LIN {X 0,Y 467.107,Z 376.18,A -85,B 0,C 180,E1 -7634.539,E2 -7634.539} C_VEL
LIN {X 0,Y 467.124,Z 376.451,A -85,B 0,C 180,E1 -7634.607,E2 -7634.607} C_VEL
LIN {X 0,Y 469.476,Z 389.998,A -85,B 0,C 180,E1 -7635.044,E2 -7635.044} C_VEL
LIN {X 0,Y 470.129,Z 395.713,A -85,B 0,C 180,E1 -7635.278,E2 -7635.278} C_VEL
LIN {X 0,Y 469.712,Z 407.365,A -85,B 0,C 180,E1 -7635.818,E2 -7635.818} C_VEL
LIN {X 0,Y 469.278,Z 418.568,A -85,B 0,C 180,E1 -7636.5,E2 -7636.5} C_VEL
LIN {X 0,Y 468.844,Z 429.048,A -85,B 0,C 180,E1 -7637.305,E2 -7637.305} C_VEL
LIN {X 0,Y 468.368,Z 439.611,A -85,B 0,C 180,E1 -7638.312,E2 -7638.312} C_VEL
LIN {X 0,Y 467.876,Z 448.784,A -85,B 0,C 180,E1 -7639.397,E2 -7639.397} C_VEL
LIN {X 0,Y 467.447,Z 457.686,A -85,B 0,C 180,E1 -7640.699,E2 -7640.699} C_VEL
LIN {X 0,Y 467.093,Z 464.847,A -85,B 0,C 180,E1 -7641.999,E2 -7641.999} C_VEL
LIN {X 0,Y 466.908,Z 471.07,A -85,B 0,C 180,E1 -7643.438,E2 -7643.438} C_VEL
LIN {X 0,Y 466.784,Z 475.676,A -85,B 0,C 180,E1 -7644.817,E2 -7644.817} C_VEL
LIN {X 0,Y 466.663,Z 477.957,A -85,B 0,C 180,E1 -7645.681,E2 -7645.681} C_VEL
LIN {X 0,Y 466.695,Z 479.806,A -85,B 0,C 180,E1 -7646.546,E2 -7646.546} C_VEL
LIN {X 0,Y 466.646,Z 481.192,A -85,B 0,C 180,E1 -7647.41,E2 -7647.41} C_VEL
LIN {X 0,Y 466.589,Z 482.785,A -85,B 0,C 180,E1 -7649.137,E2 -7649.137} C_VEL
LIN {X 0,Y 466.57,Z 483,A -85,B 0,C 180,E1 -7650,E2 -7650} C_VEL
LIN {X 0,Y 466.589,Z 482.786,A -85,B 0,C 180,E1 -7650.863,E2 -7650.863} C_VEL
LIN {X 0,Y 466.646,Z 481.196,A -85,B 0,C 180,E1 -7652.589,E2 -7652.589} C_VEL
LIN {X 0,Y 466.695,Z 479.811,A -85,B 0,C 180,E1 -7653.453,E2 -7653.453} C_VEL
LIN {X 0,Y 466.703,Z 476.896,A -85,B 0,C 180,E1 -7654.75,E2 -7654.75} C_VEL
LIN {X 0,Y 466.84,Z 472.949,A -85,B 0,C 180,E1 -7656.049,E2 -7656.049} C_VEL
LIN {X 0,Y 466.998,Z 466.878,A -85,B 0,C 180,E1 -7657.566,E2 -7657.566} C_VEL
LIN {X 0,Y 467.349,Z 460.238,A -85,B 0,C 180,E1 -7658.866,E2 -7658.866} C_VEL
LIN {X 0,Y 467.738,Z 451.996,A -85,B 0,C 180,E1 -7660.168,E2 -7660.168} C_VEL
LIN {X 0,Y 468.133,Z 443.527,A -85,B 0,C 180,E1 -7661.254,E2 -7661.254} C_VEL
LIN {X 0,Y 468.659,Z 433.246,A -85,B 0,C 180,E1 -7662.319,E2 -7662.319} C_VEL
LIN {X 0,Y 469.104,Z 421.661,A -85,B 0,C 180,E1 -7663.284,E2 -7663.284} C_VEL
LIN {X 0,Y 469.629,Z 409.366,A -85,B 0,C 180,E1 -7664.074,E2 -7664.074} C_VEL
LIN {X 0,Y 470.056,Z 397.023,A -85,B 0,C 180,E1 -7664.669,E2 -7664.669} C_VEL
LIN {X 0,Y 469.836,Z 392.579,A -85,B 0,C 180,E1 -7664.85,E2 -7664.85} C_VEL
LIN {X 0,Y 467.621,Z 379.497,A -85,B 0,C 180,E1 -7665.312,E2 -7665.312} C_VEL
LIN {X 0,Y 467.094,Z 376.299,A -85,B 0,C 180,E1 -7665.407,E2 -7665.407} C_VEL
LIN {X 0,Y 467.229,Z 368.194,A -85,B 0,C 180,E1 -7668.623,E2 -7668.623} C_VEL
LIN {X 0,Y 467.418,Z 360.751,A -85,B 0,C 180,E1 -7671.614,E2 -7671.614} C_VEL
LIN {X 0,Y 467.623,Z 353.969,A -85,B 0,C 180,E1 -7674.412,E2 -7674.412} C_VEL
LIN {X 0,Y 467.938,Z 346.089,A -85,B 0,C 180,E1 -7677.747,E2 -7677.747} C_VEL
LIN {X 0,Y 468.177,Z 339.319,A -85,B 0,C 180,E1 -7680.689,E2 -7680.689} C_VEL
LIN {X 0,Y 468.481,Z 332.557,A -85,B 0,C 180,E1 -7683.714,E2 -7683.714} C_VEL
LIN {X 0,Y 468.553,Z 327.839,A -85,B 0,C 180,E1 -7685.907,E2 -7685.907} C_VEL
LIN {X 0,Y 467.811,Z 322.365,A -85,B 0,C 180,E1 -7688.629,E2 -7688.629} C_VEL
LIN {X 0,Y 467.615,Z 321.24,A -85,B 0,C 180,E1 -7689.279,E2 -7689.279} C_VEL
LIN {X 0,Y 467.614,Z 321.241,A -85,B 0,C 180,E1 -7692.57,E2 -7692.57} C_VEL
LIN {X 0,Y 467.564,Z 321.245,A -85,B 0,C 180,E1 -7695.052,E2 -7695.052} C_VEL
LIN {X 0,Y 467.558,Z 321.246,A -85,B 0,C 180,E1 -7698.724,E2 -7698.724} C_VEL
LIN {X 0,Y 467.558,Z 321.243,A -85,B 0,C 180,E1 -7701.955,E2 -7701.955} C_VEL
LIN {X 0,Y 467.561,Z 321.244,A -85,B 0,C 180,E1 -7705.167,E2 -7705.167} C_VEL
LIN {X 0,Y 467.573,Z 321.242,A -85,B 0,C 180,E1 -7708.259,E2 -7708.259} C_VEL
LIN {X 0,Y 467.536,Z 321.245,A -85,B 0,C 180,E1 -7711.248,E2 -7711.248} C_VEL
LIN {X 0,Y 467.584,Z 321.244,A -85,B 0,C 180,E1 -7714.396,E2 -7714.396} C_VEL
LIN {X 0,Y 467.568,Z 321.242,A -85,B 0,C 180,E1 -7716.995,E2 -7716.995} C_VEL
LIN {X 0,Y 467.614,Z 321.239,A -85,B 0,C 180,E1 -7719.777,E2 -7719.777} C_VEL
LIN {X 0,Y 467.597,Z 321.241,A -85,B 0,C 180,E1 -7722.506,E2 -7722.506} C_VEL
LIN {X 0,Y 467.589,Z 321.239,A -85,B 0,C 180,E1 -7725.196,E2 -7725.196} C_VEL
LIN {X 0,Y 467.645,Z 321.235,A -85,B 0,C 180,E1 -7727.854,E2 -7727.854} C_VEL
LIN {X 0,Y 467.672,Z 321.23,A -85,B 0,C 180,E1 -7731.357,E2 -7731.357} C_VEL
LIN {X 0,Y 467.744,Z 321.221,A -85,B 0,C 180,E1 -7733.963,E2 -7733.963} C_VEL
LIN {X 0,Y 467.849,Z 321.208,A -85,B 0,C 180,E1 -7737.417,E2 -7737.417} C_VEL
LIN {X 0,Y 467.866,Z 321.207,A -85,B 0,C 180,E1 -7740,E2 -7740} C_VEL
LIN {X 0,Y 467.849,Z 321.205,A -85,B 0,C 180,E1 -7742.583,E2 -7742.583} C_VEL
LIN {X 0,Y 467.74,Z 321.221,A -85,B 0,C 180,E1 -7746.037,E2 -7746.037} C_VEL
LIN {X 0,Y 467.672,Z 321.23,A -85,B 0,C 180,E1 -7748.643,E2 -7748.643} C_VEL
LIN {X 0,Y 467.645,Z 321.233,A -85,B 0,C 180,E1 -7752.146,E2 -7752.146} C_VEL
LIN {X 0,Y 467.639,Z 321.232,A -85,B 0,C 180,E1 -7755.885,E2 -7755.885} C_VEL
LIN {X 0,Y 467.615,Z 321.238,A -85,B 0,C 180,E1 -7759.308,E2 -7759.308} C_VEL
LIN {X 0,Y 467.526,Z 321.248,A -85,B 0,C 180,E1 -7762.074,E2 -7762.074} C_VEL
LIN {X 0,Y 467.574,Z 321.242,A -85,B 0,C 180,E1 -7764.889,E2 -7764.889} C_VEL
LIN {X 0,Y 467.552,Z 321.244,A -85,B 0,C 180,E1 -7767.774,E2 -7767.774} C_VEL
LIN {X 0,Y 467.557,Z 321.245,A -85,B 0,C 180,E1 -7771.045,E2 -7771.045} C_VEL
LIN {X 0,Y 467.583,Z 321.242,A -85,B 0,C 180,E1 -7774.243,E2 -7774.243} C_VEL
LIN {X 0,Y 467.543,Z 321.247,A -85,B 0,C 180,E1 -7777.188,E2 -7777.188} C_VEL
LIN {X 0,Y 467.551,Z 321.245,A -85,B 0,C 180,E1 -7780.268,E2 -7780.268} C_VEL
LIN {X 0,Y 467.54,Z 321.244,A -85,B 0,C 180,E1 -7783.747,E2 -7783.747} C_VEL
LIN {X 0,Y 467.549,Z 321.247,A -85,B 0,C 180,E1 -7786.256,E2 -7786.256} C_VEL
LIN {X 0,Y 467.581,Z 321.241,A -85,B 0,C 180,E1 -7788.723,E2 -7788.723} C_VEL
LIN {X 0,Y 467.569,Z 321.243,A -85,B 0,C 180,E1 -7791.408,E2 -7791.408} C_VEL
LIN {X 0,Y 467.462,Z 321.257,A -85,B 0,C 180,E1 -7794.278,E2 -7794.278} C_VEL
LIN {X 0,Y 467.518,Z 322.884,A -85,B 0,C 180,E1 -7795.771,E2 -7795.771} C_VEL
LIN {X 0,Y 467.362,Z 327.675,A -85,B 0,C 180,E1 -7799.252,E2 -7799.252} C_VEL
LIN {X 0,Y 467.182,Z 331.852,A -85,B 0,C 180,E1 -7802.204,E2 -7802.204} C_VEL
LIN {X 0,Y 467.124,Z 335.994,A -85,B 0,C 180,E1 -7805.086,E2 -7805.086} C_VEL
LIN {X 0,Y 466.969,Z 340.133,A -85,B 0,C 180,E1 -7807.899,E2 -7807.899} C_VEL
LIN {X 0,Y 466.889,Z 344.326,A -85,B 0,C 180,E1 -7810.661,E2 -7810.661} C_VEL
LIN {X 0,Y 466.806,Z 349.167,A -85,B 0,C 180,E1 -7813.739,E2 -7813.739} C_VEL
LIN {X 0,Y 466.72,Z 350.349,A -85,B 0,C 180,E1 -7814.072,E2 -7814.072} C_VEL
LIN {X 0,Y 466.388,Z 353.156,A -85,B 0,C 180,E1 -7814.423,E2 -7814.423} C_VEL
LIN {X 0,Y 465.742,Z 357.77,A -85,B 0,C 180,E1 -7814.736,E2 -7814.736} C_VEL
LIN {X 0,Y 464.822,Z 363.833,A -85,B 0,C 180,E1 -7814.982,E2 -7814.982} C_VEL
LIN {X 0,Y 463.865,Z 370.07,A -85,B 0,C 180,E1 -7815.197,E2 -7815.197} C_VEL
LIN {X 0,Y 463.117,Z 377.21,A -85,B 0,C 180,E1 -7815.509,E2 -7815.509} C_VEL
LIN {X 0,Y 462.623,Z 388.395,A -85,B 0,C 180,E1 -7816.158,E2 -7816.158} C_VEL
LIN {X 0,Y 462.173,Z 400.091,A -85,B 0,C 180,E1 -7817.043,E2 -7817.043} C_VEL
LIN {X 0,Y 461.618,Z 410.516,A -85,B 0,C 180,E1 -7818.028,E2 -7818.028} C_VEL
LIN {X 0,Y 461.162,Z 419.064,A -85,B 0,C 180,E1 -7819.019,E2 -7819.019} C_VEL
LIN {X 0,Y 460.753,Z 426.936,A -85,B 0,C 180,E1 -7820.12,E2 -7820.12} C_VEL
LIN {X 0,Y 460.337,Z 434.631,A -85,B 0,C 180,E1 -7821.44,E2 -7821.44} C_VEL
LIN {X 0,Y 459.979,Z 441.691,A -85,B 0,C 180,E1 -7822.98,E2 -7822.98} C_VEL
LIN {X 0,Y 459.877,Z 446.391,A -85,B 0,C 180,E1 -7824.3,E2 -7824.3} C_VEL
LIN {X 0,Y 459.687,Z 449.993,A -85,B 0,C 180,E1 -7825.616,E2 -7825.616} C_VEL
LIN {X 0,Y 459.708,Z 451.852,A -85,B 0,C 180,E1 -7826.495,E2 -7826.495} C_VEL
LIN {X 0,Y 459.608,Z 453.256,A -85,B 0,C 180,E1 -7827.371,E2 -7827.371} C_VEL
LIN {X 0,Y 459.523,Z 454.869,A -85,B 0,C 180,E1 -7829.124,E2 -7829.124} C_VEL
LIN {X 0,Y 459.53,Z 455.103,A -85,B 0,C 180,E1 -7830,E2 -7830} C_VEL
LIN {X 0,Y 459.523,Z 454.917,A -85,B 0,C 180,E1 -7830.877,E2 -7830.877} C_VEL
LIN {X 0,Y 459.608,Z 453.367,A -85,B 0,C 180,E1 -7832.63,E2 -7832.63} C_VEL
LIN {X 0,Y 459.708,Z 452.012,A -85,B 0,C 180,E1 -7833.506,E2 -7833.506} C_VEL
LIN {X 0,Y 459.674,Z 449.153,A -85,B 0,C 180,E1 -7834.824,E2 -7834.824} C_VEL
LIN {X 0,Y 459.939,Z 445.267,A -85,B 0,C 180,E1 -7836.14,E2 -7836.14} C_VEL
LIN {X 0,Y 460.051,Z 440.261,A -85,B 0,C 180,E1 -7837.461,E2 -7837.461} C_VEL
LIN {X 0,Y 460.379,Z 433.956,A -85,B 0,C 180,E1 -7838.781,E2 -7838.781} C_VEL
LIN {X 0,Y 460.768,Z 426.061,A -85,B 0,C 180,E1 -7840.103,E2 -7840.103} C_VEL
LIN {X 0,Y 461.175,Z 418.013,A -85,B 0,C 180,E1 -7841.204,E2 -7841.204} C_VEL
LIN {X 0,Y 461.799,Z 408.186,A -85,B 0,C 180,E1 -7842.302,E2 -7842.302} C_VEL
LIN {X 0,Y 462.179,Z 398.523,A -85,B 0,C 180,E1 -7843.185,E2 -7843.185} C_VEL
LIN {X 0,Y 462.632,Z 388.238,A -85,B 0,C 180,E1 -7843.944,E2 -7843.944} C_VEL
LIN {X 0,Y 463.138,Z 376.598,A -85,B 0,C 180,E1 -7844.613,E2 -7844.613} C_VEL
LIN {X 0,Y 463.284,Z 367.958,A -85,B 0,C 180,E1 -7845.007,E2 -7845.007} C_VEL
LIN {X 0,Y 460.888,Z 355.74,A -85,B 0,C 180,E1 -7845.503,E2 -7845.503} C_VEL
LIN {X 0,Y 459.767,Z 350.859,A -85,B 0,C 180,E1 -7845.672,E2 -7845.672} C_VEL
LIN {X 0,Y 459.831,Z 346.077,A -85,B 0,C 180,E1 -7848.721,E2 -7848.721} C_VEL
LIN {X 0,Y 459.901,Z 341.846,A -85,B 0,C 180,E1 -7851.516,E2 -7851.516} C_VEL
LIN {X 0,Y 460.006,Z 337.676,A -85,B 0,C 180,E1 -7854.362,E2 -7854.362} C_VEL
LIN {X 0,Y 460.132,Z 333.012,A -85,B 0,C 180,E1 -7857.639,E2 -7857.639} C_VEL
LIN {X 0,Y 460.26,Z 329.333,A -85,B 0,C 180,E1 -7860.258,E2 -7860.258} C_VEL
LIN {X 0,Y 460.403,Z 325.125,A -85,B 0,C 180,E1 -7863.335,E2 -7863.335} C_VEL
LIN {X 0,Y 460.415,Z 322.298,A -85,B 0,C 180,E1 -7865.454,E2 -7865.454} C_VEL
LIN {X 0,Y 460.497,Z 322.124,A -85,B 0,C 180,E1 -7867.623,E2 -7867.623} C_VEL
LIN {X 0,Y 460.539,Z 322.119,A -85,B 0,C 180,E1 -7870.269,E2 -7870.269} C_VEL
LIN {X 0,Y 460.498,Z 322.124,A -85,B 0,C 180,E1 -7873.375,E2 -7873.375} C_VEL
LIN {X 0,Y 460.494,Z 322.122,A -85,B 0,C 180,E1 -7876.624,E2 -7876.624} C_VEL
LIN {X 0,Y 460.521,Z 322.121,A -85,B 0,C 180,E1 -7879.733,E2 -7879.733} C_VEL
LIN {X 0,Y 460.498,Z 322.123,A -85,B 0,C 180,E1 -7882.523,E2 -7882.523} C_VEL
LIN {X 0,Y 460.546,Z 322.12,A -85,B 0,C 180,E1 -7885.624,E2 -7885.624} C_VEL
LIN {X 0,Y 460.534,Z 322.118,A -85,B 0,C 180,E1 -7888.744,E2 -7888.744} C_VEL
LIN {X 0,Y 460.527,Z 322.118,A -85,B 0,C 180,E1 -7892.266,E2 -7892.266} C_VEL
LIN {X 0,Y 460.521,Z 322.123,A -85,B 0,C 180,E1 -7894.703,E2 -7894.703} C_VEL
LIN {X 0,Y 460.506,Z 322.123,A -85,B 0,C 180,E1 -7897.571,E2 -7897.571} C_VEL
LIN {X 0,Y 460.566,Z 322.114,A -85,B 0,C 180,E1 -7900.384,E2 -7900.384} C_VEL
LIN {X 0,Y 460.559,Z 322.116,A -85,B 0,C 180,E1 -7903.146,E2 -7903.146} C_VEL
LIN {X 0,Y 460.542,Z 322.116,A -85,B 0,C 180,E1 -7905.867,E2 -7905.867} C_VEL
LIN {X 0,Y 460.606,Z 322.111,A -85,B 0,C 180,E1 -7908.559,E2 -7908.559} C_VEL
LIN {X 0,Y 460.691,Z 322.1,A -85,B 0,C 180,E1 -7912.108,E2 -7912.108} C_VEL
LIN {X 0,Y 460.694,Z 322.102,A -85,B 0,C 180,E1 -7914.748,E2 -7914.748} C_VEL
LIN {X 0,Y 460.795,Z 322.083,A -85,B 0,C 180,E1 -7917.377,E2 -7917.377} C_VEL
LIN {X 0,Y 460.84,Z 322.082,A -85,B 0,C 180,E1 -7920,E2 -7920} C_VEL
LIN {X 0,Y 460.794,Z 322.087,A -85,B 0,C 180,E1 -7922.622,E2 -7922.622} C_VEL
LIN {X 0,Y 460.707,Z 322.098,A -85,B 0,C 180,E1 -7926.13,E2 -7926.13} C_VEL
LIN {X 0,Y 460.625,Z 322.107,A -85,B 0,C 180,E1 -7928.776,E2 -7928.776} C_VEL
LIN {X 0,Y 460.604,Z 322.11,A -85,B 0,C 180,E1 -7932.334,E2 -7932.334} C_VEL
LIN {X 0,Y 460.596,Z 322.112,A -85,B 0,C 180,E1 -7935.998,E2 -7935.998} C_VEL
LIN {X 0,Y 460.567,Z 322.115,A -85,B 0,C 180,E1 -7938.902,E2 -7938.902} C_VEL
LIN {X 0,Y 460.512,Z 322.122,A -85,B 0,C 180,E1 -7941.486,E2 -7941.486} C_VEL
LIN {X 0,Y 460.526,Z 322.119,A -85,B 0,C 180,E1 -7944.333,E2 -7944.333} C_VEL
LIN {X 0,Y 460.51,Z 322.122,A -85,B 0,C 180,E1 -7947.248,E2 -7947.248} C_VEL
LIN {X 0,Y 460.5,Z 322.123,A -85,B 0,C 180,E1 -7950.241,E2 -7950.241} C_VEL
LIN {X 0,Y 460.527,Z 322.12,A -85,B 0,C 180,E1 -7953.325,E2 -7953.325} C_VEL
LIN {X 0,Y 460.476,Z 322.126,A -85,B 0,C 180,E1 -7956.53,E2 -7956.53} C_VEL
LIN {X 0,Y 460.502,Z 322.122,A -85,B 0,C 180,E1 -7958.892,E2 -7958.892} C_VEL
LIN {X 0,Y 460.499,Z 322.123,A -85,B 0,C 180,E1 -7961.599,E2 -7961.599} C_VEL
LIN {X 0,Y 460.509,Z 322.126,A -85,B 0,C 180,E1 -7964.59,E2 -7964.59} C_VEL
LIN {X 0,Y 460.522,Z 322.123,A -85,B 0,C 180,E1 -7967.819,E2 -7967.819} C_VEL
LIN {X 0,Y 460.594,Z 322.299,A -85,B 0,C 180,E1 -7970.65,E2 -7970.65} C_VEL
LIN {X 0,Y 461.487,Z 327.991,A -85,B 0,C 180,E1 -7973.564,E2 -7973.564} C_VEL
LIN {X 0,Y 461.51,Z 332.461,A -85,B 0,C 180,E1 -7975.706,E2 -7975.706} C_VEL
LIN {X 0,Y 461.231,Z 339.206,A -85,B 0,C 180,E1 -7978.797,E2 -7978.797} C_VEL
LIN {X 0,Y 460.924,Z 346.84,A -85,B 0,C 180,E1 -7982.173,E2 -7982.173} C_VEL
LIN {X 0,Y 460.606,Z 353.852,A -85,B 0,C 180,E1 -7985.191,E2 -7985.191} C_VEL
LIN {X 0,Y 460.389,Z 360.659,A -85,B 0,C 180,E1 -7988.037,E2 -7988.037} C_VEL
LIN {X 0,Y 460.175,Z 368.613,A -85,B 0,C 180,E1 -7991.293,E2 -7991.293} C_VEL
LIN {X 0,Y 460.04,Z 376.143,A -85,B 0,C 180,E1 -7994.353,E2 -7994.353} C_VEL
LIN {X 0,Y 462.464,Z 390.155,A -85,B 0,C 180,E1 -7994.826,E2 -7994.826} C_VEL
LIN {X 0,Y 463.206,Z 396.8,A -85,B 0,C 180,E1 -7995.109,E2 -7995.109} C_VEL
LIN {X 0,Y 462.727,Z 409.139,A -85,B 0,C 180,E1 -7995.711,E2 -7995.711} C_VEL
LIN {X 0,Y 462.223,Z 421.008,A -85,B 0,C 180,E1 -7996.481,E2 -7996.481} C_VEL
LIN {X 0,Y 461.719,Z 432.146,A -85,B 0,C 180,E1 -7997.409,E2 -7997.409} C_VEL
LIN {X 0,Y 461.259,Z 441.353,A -85,B 0,C 180,E1 -7998.353,E2 -7998.353} C_VEL
LIN {X 0,Y 460.756,Z 450.206,A -85,B 0,C 180,E1 -7999.453,E2 -7999.453} C_VEL
LIN {X 0,Y 460.346,Z 458.842,A -85,B 0,C 180,E1 -8000.775,E2 -8000.775} C_VEL
LIN {X 0,Y 459.98,Z 465.743,A -85,B 0,C 180,E1 -8002.096,E2 -8002.096} C_VEL
LIN {X 0,Y 459.808,Z 471.46,A -85,B 0,C 180,E1 -8003.467,E2 -8003.467} C_VEL
LIN {X 0,Y 459.701,Z 475.619,A -85,B 0,C 180,E1 -8004.737,E2 -8004.737} C_VEL
LIN {X 0,Y 459.58,Z 477.914,A -85,B 0,C 180,E1 -8005.615,E2 -8005.615} C_VEL
LIN {X 0,Y 459.591,Z 479.778,A -85,B 0,C 180,E1 -8006.493,E2 -8006.493} C_VEL
LIN {X 0,Y 459.57,Z 481.175,A -85,B 0,C 180,E1 -8007.37,E2 -8007.37} C_VEL
LIN {X 0,Y 459.494,Z 482.778,A -85,B 0,C 180,E1 -8009.123,E2 -8009.123} C_VEL
LIN {X 0,Y 459.474,Z 482.994,A -85,B 0,C 180,E1 -8010,E2 -8010} C_VEL
LIN {X 0,Y 459.494,Z 482.779,A -85,B 0,C 180,E1 -8010.876,E2 -8010.876} C_VEL
LIN {X 0,Y 459.57,Z 481.179,A -85,B 0,C 180,E1 -8012.629,E2 -8012.629} C_VEL
LIN {X 0,Y 459.591,Z 479.783,A -85,B 0,C 180,E1 -8013.506,E2 -8013.506} C_VEL
LIN {X 0,Y 459.634,Z 476.847,A -85,B 0,C 180,E1 -8014.824,E2 -8014.824} C_VEL
LIN {X 0,Y 459.757,Z 472.873,A -85,B 0,C 180,E1 -8016.142,E2 -8016.142} C_VEL
LIN {X 0,Y 459.928,Z 466.76,A -85,B 0,C 180,E1 -8017.683,E2 -8017.683} C_VEL
LIN {X 0,Y 460.305,Z 460.085,A -85,B 0,C 180,E1 -8019.003,E2 -8019.003} C_VEL
LIN {X 0,Y 460.7,Z 451.799,A -85,B 0,C 180,E1 -8020.325,E2 -8020.325} C_VEL
LIN {X 0,Y 461.144,Z 443.31,A -85,B 0,C 180,E1 -8021.427,E2 -8021.427} C_VEL
LIN {X 0,Y 461.674,Z 433.197,A -85,B 0,C 180,E1 -8022.492,E2 -8022.492} C_VEL
LIN {X 0,Y 462.119,Z 422.733,A -85,B 0,C 180,E1 -8023.387,E2 -8023.387} C_VEL
LIN {X 0,Y 462.648,Z 411.072,A -85,B 0,C 180,E1 -8024.178,E2 -8024.178} C_VEL
LIN {X 0,Y 463.128,Z 399.413,A -85,B 0,C 180,E1 -8024.781,E2 -8024.781} C_VEL
LIN {X 0,Y 462.969,Z 393.828,A -85,B 0,C 180,E1 -8025.022,E2 -8025.022} C_VEL
LIN {X 0,Y 460.806,Z 380.747,A -85,B 0,C 180,E1 -8025.508,E2 -8025.508} C_VEL
LIN {X 0,Y 460.028,Z 376.103,A -85,B 0,C 180,E1 -8025.666,E2 -8025.666} C_VEL
LIN {X 0,Y 460.197,Z 367.545,A -85,B 0,C 180,E1 -8029.121,E2 -8029.121} C_VEL
LIN {X 0,Y 460.424,Z 359.456,A -85,B 0,C 180,E1 -8032.432,E2 -8032.432} C_VEL
LIN {X 0,Y 460.735,Z 351.428,A -85,B 0,C 180,E1 -8035.844,E2 -8035.844} C_VEL
LIN {X 0,Y 460.981,Z 344.842,A -85,B 0,C 180,E1 -8038.7,E2 -8038.7} C_VEL
LIN {X 0,Y 461.246,Z 338.699,A -85,B 0,C 180,E1 -8041.43,E2 -8041.43} C_VEL
LIN {X 0,Y 461.55,Z 331.611,A -85,B 0,C 180,E1 -8044.689,E2 -8044.689} C_VEL
LIN {X 0,Y 461.49,Z 327.978,A -85,B 0,C 180,E1 -8046.435,E2 -8046.435} C_VEL
LIN {X 0,Y 460.593,Z 322.114,A -85,B 0,C 180,E1 -8049.477,E2 -8049.477} C_VEL
LIN {X 0,Y 460.538,Z 322.122,A -85,B 0,C 180,E1 -8052.903,E2 -8052.903} C_VEL
LIN {X 0,Y 460.5,Z 322.124,A -85,B 0,C 180,E1 -8055.83,E2 -8055.83} C_VEL
LIN {X 0,Y 460.511,Z 322.123,A -85,B 0,C 180,E1 -8058.986,E2 -8058.986} C_VEL
LIN {X 0,Y 460.52,Z 322.124,A -85,B 0,C 180,E1 -8062.519,E2 -8062.519} C_VEL
LIN {X 0,Y 460.541,Z 322.118,A -85,B 0,C 180,E1 -8065.623,E2 -8065.623} C_VEL
LIN {X 0,Y 460.529,Z 322.122,A -85,B 0,C 180,E1 -8068.744,E2 -8068.744} C_VEL
LIN {X 0,Y 460.522,Z 322.121,A -85,B 0,C 180,E1 -8072.265,E2 -8072.265} C_VEL
LIN {X 0,Y 460.53,Z 322.119,A -85,B 0,C 180,E1 -8074.704,E2 -8074.704} C_VEL
LIN {X 0,Y 460.503,Z 322.122,A -85,B 0,C 180,E1 -8077.571,E2 -8077.571} C_VEL
LIN {X 0,Y 460.56,Z 322.116,A -85,B 0,C 180,E1 -8080.384,E2 -8080.384} C_VEL
LIN {X 0,Y 460.554,Z 322.116,A -85,B 0,C 180,E1 -8083.146,E2 -8083.146} C_VEL
LIN {X 0,Y 460.537,Z 322.119,A -85,B 0,C 180,E1 -8085.867,E2 -8085.867} C_VEL
LIN {X 0,Y 460.6,Z 322.109,A -85,B 0,C 180,E1 -8088.559,E2 -8088.559} C_VEL
LIN {X 0,Y 460.685,Z 322.1,A -85,B 0,C 180,E1 -8092.108,E2 -8092.108} C_VEL
LIN {X 0,Y 460.696,Z 322.098,A -85,B 0,C 180,E1 -8094.748,E2 -8094.748} C_VEL
LIN {X 0,Y 460.814,Z 322.084,A -85,B 0,C 180,E1 -8097.378,E2 -8097.378} C_VEL
LIN {X 0,Y 460.836,Z 322.083,A -85,B 0,C 180,E1 -8100,E2 -8100} C_VEL
LIN {X 0,Y 460.79,Z 322.084,A -85,B 0,C 180,E1 -8102.623,E2 -8102.623} C_VEL
LIN {X 0,Y 460.705,Z 322.097,A -85,B 0,C 180,E1 -8106.13,E2 -8106.13} C_VEL
LIN {X 0,Y 460.619,Z 322.109,A -85,B 0,C 180,E1 -8108.776,E2 -8108.776} C_VEL
LIN {X 0,Y 460.598,Z 322.11,A -85,B 0,C 180,E1 -8112.335,E2 -8112.335} C_VEL
LIN {X 0,Y 460.59,Z 322.109,A -85,B 0,C 180,E1 -8115.998,E2 -8115.998} C_VEL
LIN {X 0,Y 460.562,Z 322.118,A -85,B 0,C 180,E1 -8118.902,E2 -8118.902} C_VEL
LIN {X 0,Y 460.507,Z 322.122,A -85,B 0,C 180,E1 -8121.486,E2 -8121.486} C_VEL
LIN {X 0,Y 460.52,Z 322.121,A -85,B 0,C 180,E1 -8124.334,E2 -8124.334} C_VEL
LIN {X 0,Y 460.508,Z 322.125,A -85,B 0,C 180,E1 -8127.248,E2 -8127.248} C_VEL
LIN {X 0,Y 460.495,Z 322.121,A -85,B 0,C 180,E1 -8130.241,E2 -8130.241} C_VEL
LIN {X 0,Y 460.522,Z 322.119,A -85,B 0,C 180,E1 -8133.326,E2 -8133.326} C_VEL
LIN {X 0,Y 460.472,Z 322.128,A -85,B 0,C 180,E1 -8136.53,E2 -8136.53} C_VEL
LIN {X 0,Y 460.507,Z 322.122,A -85,B 0,C 180,E1 -8139.865,E2 -8139.865} C_VEL
LIN {X 0,Y 460.473,Z 322.128,A -85,B 0,C 180,E1 -8142.897,E2 -8142.897} C_VEL
LIN {X 0,Y 460.504,Z 322.121,A -85,B 0,C 180,E1 -8145.832,E2 -8145.832} C_VEL
LIN {X 0,Y 460.535,Z 322.119,A -85,B 0,C 180,E1 -8148.991,E2 -8148.991} C_VEL
LIN {X 0,Y 460.539,Z 322.118,A -85,B 0,C 180,E1 -8151.27,E2 -8151.27} C_VEL
LIN {X 0,Y 460.385,Z 322.175,A -85,B 0,C 180,E1 -8154.545,E2 -8154.545} C_VEL
LIN {X 0,Y 460.398,Z 325.568,A -85,B 0,C 180,E1 -8157.096,E2 -8157.096} C_VEL
LIN {X 0,Y 460.262,Z 329.196,A -85,B 0,C 180,E1 -8159.743,E2 -8159.743} C_VEL
LIN {X 0,Y 460.122,Z 333.372,A -85,B 0,C 180,E1 -8162.728,E2 -8162.728} C_VEL
LIN {X 0,Y 460.047,Z 337.537,A -85,B 0,C 180,E1 -8165.641,E2 -8165.641} C_VEL
LIN {X 0,Y 459.907,Z 342.129,A -85,B 0,C 180,E1 -8168.775,E2 -8168.775} C_VEL
LIN {X 0,Y 459.782,Z 347.341,A -85,B 0,C 180,E1 -8172.2,E2 -8172.2} C_VEL
LIN {X 0,Y 459.814,Z 350.87,A -85,B 0,C 180,E1 -8174.429,E2 -8174.429} C_VEL
LIN {X 0,Y 462.721,Z 364.62,A -85,B 0,C 180,E1 -8174.939,E2 -8174.939} C_VEL
LIN {X 0,Y 463.319,Z 369.874,A -85,B 0,C 180,E1 -8175.169,E2 -8175.169} C_VEL
LIN {X 0,Y 463.117,Z 377.21,A -85,B 0,C 180,E1 -8175.509,E2 -8175.509} C_VEL
LIN {X 0,Y 462.311,Z 382.642,A -85,B 0,C 180,E1 -8175.779,E2 -8175.779} C_VEL
LIN {X 0,Y 459.222,Z 391.298,A -85,B 0,C 180,E1 -8176.239,E2 -8176.239} C_VEL
LIN {X 0,Y 456.032,Z 399.557,A -85,B 0,C 180,E1 -8176.794,E2 -8176.794} C_VEL
LIN {X 0,Y 455.075,Z 404.364,A -85,B 0,C 180,E1 -8177.206,E2 -8177.206} C_VEL
LIN {X 0,Y 454.567,Z 413.753,A -85,B 0,C 180,E1 -8178.18,E2 -8178.18} C_VEL
LIN {X 0,Y 454.044,Z 422.597,A -85,B 0,C 180,E1 -8179.296,E2 -8179.296} C_VEL
LIN {X 0,Y 453.543,Z 431.224,A -85,B 0,C 180,E1 -8180.637,E2 -8180.637} C_VEL
LIN {X 0,Y 453.115,Z 438.1,A -85,B 0,C 180,E1 -8181.976,E2 -8181.976} C_VEL
LIN {X 0,Y 452.879,Z 443.572,A -85,B 0,C 180,E1 -8183.308,E2 -8183.308} C_VEL
LIN {X 0,Y 452.697,Z 447.924,A -85,B 0,C 180,E1 -8184.656,E2 -8184.656} C_VEL
LIN {X 0,Y 452.595,Z 450.21,A -85,B 0,C 180,E1 -8185.547,E2 -8185.547} C_VEL
LIN {X 0,Y 452.624,Z 452.068,A -85,B 0,C 180,E1 -8186.44,E2 -8186.44} C_VEL
LIN {X 0,Y 452.535,Z 453.472,A -85,B 0,C 180,E1 -8187.33,E2 -8187.33} C_VEL
LIN {X 0,Y 452.431,Z 455.084,A -85,B 0,C 180,E1 -8189.11,E2 -8189.11} C_VEL
LIN {X 0,Y 452.435,Z 455.319,A -85,B 0,C 180,E1 -8190,E2 -8190} C_VEL
LIN {X 0,Y 452.431,Z 455.132,A -85,B 0,C 180,E1 -8190.89,E2 -8190.89} C_VEL
LIN {X 0,Y 452.535,Z 453.582,A -85,B 0,C 180,E1 -8192.671,E2 -8192.671} C_VEL
LIN {X 0,Y 452.623,Z 452.226,A -85,B 0,C 180,E1 -8193.561,E2 -8193.561} C_VEL
LIN {X 0,Y 452.605,Z 449.367,A -85,B 0,C 180,E1 -8194.9,E2 -8194.9} C_VEL
LIN {X 0,Y 452.864,Z 445.482,A -85,B 0,C 180,E1 -8196.237,E2 -8196.237} C_VEL
LIN {X 0,Y 452.995,Z 440.475,A -85,B 0,C 180,E1 -8197.578,E2 -8197.578} C_VEL
LIN {X 0,Y 453.369,Z 434.169,A -85,B 0,C 180,E1 -8198.918,E2 -8198.918} C_VEL
LIN {X 0,Y 453.768,Z 426.274,A -85,B 0,C 180,E1 -8200.26,E2 -8200.26} C_VEL
LIN {X 0,Y 454.34,Z 416.45,A -85,B 0,C 180,E1 -8201.601,E2 -8201.601} C_VEL
LIN {X 0,Y 454.998,Z 406.369,A -85,B 0,C 180,E1 -8202.693,E2 -8202.693} C_VEL
LIN {X 0,Y 455.401,Z 395.936,A -85,B 0,C 180,E1 -8203.612,E2 -8203.612} C_VEL
LIN {X 0,Y 455.924,Z 384.756,A -85,B 0,C 180,E1 -8204.393,E2 -8204.393} C_VEL
LIN {X 0,Y 456.448,Z 372.184,A -85,B 0,C 180,E1 -8205.06,E2 -8205.06} C_VEL
LIN {X 0,Y 456.073,Z 366.868,A -85,B 0,C 180,E1 -8205.302,E2 -8205.302} C_VEL
LIN {X 0,Y 453.381,Z 354.212,A -85,B 0,C 180,E1 -8205.81,E2 -8205.81} C_VEL
LIN {X 0,Y 452.661,Z 351.063,A -85,B 0,C 180,E1 -8205.922,E2 -8205.922} C_VEL
LIN {X 0,Y 452.771,Z 346.265,A -85,B 0,C 180,E1 -8209.024,E2 -8209.024} C_VEL
LIN {X 0,Y 452.836,Z 342.018,A -85,B 0,C 180,E1 -8211.869,E2 -8211.869} C_VEL
LIN {X 0,Y 452.963,Z 337.835,A -85,B 0,C 180,E1 -8214.766,E2 -8214.766} C_VEL
LIN {X 0,Y 453.08,Z 333.512,A -85,B 0,C 180,E1 -8217.851,E2 -8217.851} C_VEL
LIN {X 0,Y 453.247,Z 329.46,A -85,B 0,C 180,E1 -8220.777,E2 -8220.777} C_VEL
LIN {X 0,Y 453.394,Z 325.223,A -85,B 0,C 180,E1 -8223.919,E2 -8223.919} C_VEL
LIN {X 0,Y 453.391,Z 323.807,A -85,B 0,C 180,E1 -8224.997,E2 -8224.997} C_VEL
LIN {X 0,Y 453.413,Z 323.009,A -85,B 0,C 180,E1 -8226.292,E2 -8226.292} C_VEL
LIN {X 0,Y 453.467,Z 323,A -85,B 0,C 180,E1 -8229.452,E2 -8229.452} C_VEL
LIN {X 0,Y 453.476,Z 323.001,A -85,B 0,C 180,E1 -8231.934,E2 -8231.934} C_VEL
LIN {X 0,Y 453.48,Z 323,A -85,B 0,C 180,E1 -8235.471,E2 -8235.471} C_VEL
LIN {X 0,Y 453.467,Z 323.001,A -85,B 0,C 180,E1 -8239.388,E2 -8239.388} C_VEL
LIN {X 0,Y 453.451,Z 323.002,A -85,B 0,C 180,E1 -8242.81,E2 -8242.81} C_VEL
LIN {X 0,Y 453.475,Z 322.997,A -85,B 0,C 180,E1 -8246.087,E2 -8246.087} C_VEL
LIN {X 0,Y 453.471,Z 323.002,A -85,B 0,C 180,E1 -8249.24,E2 -8249.24} C_VEL
LIN {X 0,Y 453.485,Z 322.996,A -85,B 0,C 180,E1 -8252.294,E2 -8252.294} C_VEL
LIN {X 0,Y 453.486,Z 322.997,A -85,B 0,C 180,E1 -8255.264,E2 -8255.264} C_VEL
LIN {X 0,Y 453.476,Z 322.999,A -85,B 0,C 180,E1 -8258.415,E2 -8258.415} C_VEL
LIN {X 0,Y 453.518,Z 322.996,A -85,B 0,C 180,E1 -8261.008,E2 -8261.008} C_VEL
LIN {X 0,Y 453.565,Z 322.984,A -85,B 0,C 180,E1 -8263.879,E2 -8263.879} C_VEL
LIN {X 0,Y 453.559,Z 322.987,A -85,B 0,C 180,E1 -8267.471,E2 -8267.471} C_VEL
LIN {X 0,Y 453.587,Z 322.986,A -85,B 0,C 180,E1 -8271.086,E2 -8271.086} C_VEL
LIN {X 0,Y 453.674,Z 322.973,A -85,B 0,C 180,E1 -8273.775,E2 -8273.775} C_VEL
LIN {X 0,Y 453.739,Z 322.962,A -85,B 0,C 180,E1 -8277.337,E2 -8277.337} C_VEL
LIN {X 0,Y 453.809,Z 322.958,A -85,B 0,C 180,E1 -8280,E2 -8280} C_VEL
LIN {X 0,Y 453.738,Z 322.966,A -85,B 0,C 180,E1 -8282.663,E2 -8282.663} C_VEL
LIN {X 0,Y 453.674,Z 322.974,A -85,B 0,C 180,E1 -8286.225,E2 -8286.225} C_VEL
LIN {X 0,Y 453.588,Z 322.983,A -85,B 0,C 180,E1 -8288.913,E2 -8288.913} C_VEL
LIN {X 0,Y 453.559,Z 322.986,A -85,B 0,C 180,E1 -8292.529,E2 -8292.529} C_VEL
LIN {X 0,Y 453.54,Z 322.99,A -85,B 0,C 180,E1 -8296.196,E2 -8296.196} C_VEL
LIN {X 0,Y 453.516,Z 322.993,A -85,B 0,C 180,E1 -8299.041,E2 -8299.041} C_VEL
LIN {X 0,Y 453.473,Z 323,A -85,B 0,C 180,E1 -8301.836,E2 -8301.836} C_VEL
LIN {X 0,Y 453.496,Z 322.993,A -85,B 0,C 180,E1 -8304.736,E2 -8304.736} C_VEL
LIN {X 0,Y 453.471,Z 322.998,A -85,B 0,C 180,E1 -8307.946,E2 -8307.946} C_VEL
LIN {X 0,Y 453.47,Z 322.998,A -85,B 0,C 180,E1 -8310.76,E2 -8310.76} C_VEL
LIN {X 0,Y 453.475,Z 323,A -85,B 0,C 180,E1 -8313.913,E2 -8313.913} C_VEL
LIN {X 0,Y 453.468,Z 323,A -85,B 0,C 180,E1 -8317.188,E2 -8317.188} C_VEL
LIN {X 0,Y 453.467,Z 322.997,A -85,B 0,C 180,E1 -8320.612,E2 -8320.612} C_VEL
LIN {X 0,Y 453.479,Z 323.001,A -85,B 0,C 180,E1 -8324.529,E2 -8324.529} C_VEL
LIN {X 0,Y 453.479,Z 323.001,A -85,B 0,C 180,E1 -8328.21,E2 -8328.21} C_VEL
LIN {X 0,Y 453.556,Z 323.172,A -85,B 0,C 180,E1 -8330.414,E2 -8330.414} C_VEL
LIN {X 0,Y 454.484,Z 329.145,A -85,B 0,C 180,E1 -8333.525,E2 -8333.525} C_VEL
LIN {X 0,Y 454.512,Z 333.483,A -85,B 0,C 180,E1 -8335.64,E2 -8335.64} C_VEL
LIN {X 0,Y 454.223,Z 340.277,A -85,B 0,C 180,E1 -8338.807,E2 -8338.807} C_VEL
LIN {X 0,Y 453.871,Z 348.105,A -85,B 0,C 180,E1 -8342.32,E2 -8342.32} C_VEL
LIN {X 0,Y 453.557,Z 354.863,A -85,B 0,C 180,E1 -8345.268,E2 -8345.268} C_VEL
LIN {X 0,Y 453.289,Z 362.427,A -85,B 0,C 180,E1 -8348.477,E2 -8348.477} C_VEL
LIN {X 0,Y 453.123,Z 368.736,A -85,B 0,C 180,E1 -8351.106,E2 -8351.106} C_VEL
LIN {X 0,Y 452.937,Z 375.949,A -85,B 0,C 180,E1 -8354.105,E2 -8354.105} C_VEL
LIN {X 0,Y 455.387,Z 389.936,A -85,B 0,C 180,E1 -8354.585,E2 -8354.585} C_VEL
LIN {X 0,Y 456.342,Z 396.584,A -85,B 0,C 180,E1 -8354.879,E2 -8354.879} C_VEL
LIN {X 0,Y 455.831,Z 408.923,A -85,B 0,C 180,E1 -8355.49,E2 -8355.49} C_VEL
LIN {X 0,Y 455.307,Z 420.786,A -85,B 0,C 180,E1 -8356.271,E2 -8356.271} C_VEL
LIN {X 0,Y 454.782,Z 431.289,A -85,B 0,C 180,E1 -8357.152,E2 -8357.152} C_VEL
LIN {X 0,Y 454.27,Z 441.136,A -85,B 0,C 180,E1 -8358.171,E2 -8358.171} C_VEL
LIN {X 0,Y 453.736,Z 449.989,A -85,B 0,C 180,E1 -8359.288,E2 -8359.288} C_VEL
LIN {X 0,Y 453.311,Z 458.626,A -85,B 0,C 180,E1 -8360.631,E2 -8360.631} C_VEL
LIN {X 0,Y 452.924,Z 465.527,A -85,B 0,C 180,E1 -8361.972,E2 -8361.972} C_VEL
LIN {X 0,Y 452.731,Z 471.626,A -85,B 0,C 180,E1 -8363.469,E2 -8363.469} C_VEL
LIN {X 0,Y 452.567,Z 476.628,A -85,B 0,C 180,E1 -8365.1,E2 -8365.1} C_VEL
LIN {X 0,Y 452.488,Z 479.562,A -85,B 0,C 180,E1 -8366.438,E2 -8366.438} C_VEL
LIN {X 0,Y 452.496,Z 480.96,A -85,B 0,C 180,E1 -8367.329,E2 -8367.329} C_VEL
LIN {X 0,Y 452.403,Z 482.564,A -85,B 0,C 180,E1 -8369.11,E2 -8369.11} C_VEL
LIN {X 0,Y 452.381,Z 482.78,A -85,B 0,C 180,E1 -8370,E2 -8370} C_VEL
LIN {X 0,Y 452.403,Z 482.565,A -85,B 0,C 180,E1 -8370.89,E2 -8370.89} C_VEL
LIN {X 0,Y 452.496,Z 480.964,A -85,B 0,C 180,E1 -8372.67,E2 -8372.67} C_VEL
LIN {X 0,Y 452.488,Z 479.567,A -85,B 0,C 180,E1 -8373.561,E2 -8373.561} C_VEL
LIN {X 0,Y 452.567,Z 476.631,A -85,B 0,C 180,E1 -8374.899,E2 -8374.899} C_VEL
LIN {X 0,Y 452.687,Z 471.804,A -85,B 0,C 180,E1 -8376.481,E2 -8376.481} C_VEL
LIN {X 0,Y 452.926,Z 465.531,A -85,B 0,C 180,E1 -8378.027,E2 -8378.027} C_VEL
LIN {X 0,Y 453.31,Z 458.63,A -85,B 0,C 180,E1 -8379.368,E2 -8379.368} C_VEL
LIN {X 0,Y 453.736,Z 449.995,A -85,B 0,C 180,E1 -8380.711,E2 -8380.711} C_VEL
LIN {X 0,Y 454.294,Z 441.144,A -85,B 0,C 180,E1 -8381.828,E2 -8381.828} C_VEL
LIN {X 0,Y 454.835,Z 431.31,A -85,B 0,C 180,E1 -8382.844,E2 -8382.844} C_VEL
LIN {X 0,Y 455.293,Z 420.799,A -85,B 0,C 180,E1 -8383.728,E2 -8383.728} C_VEL
LIN {X 0,Y 455.846,Z 408.934,A -85,B 0,C 180,E1 -8384.508,E2 -8384.508} C_VEL
LIN {X 0,Y 456.309,Z 396.591,A -85,B 0,C 180,E1 -8385.121,E2 -8385.121} C_VEL
LIN {X 0,Y 454.37,Z 384.012,A -85,B 0,C 180,E1 -8385.642,E2 -8385.642} C_VEL
LIN {X 0,Y 452.952,Z 375.933,A -85,B 0,C 180,E1 -8385.901,E2 -8385.901} C_VEL
LIN {X 0,Y 453.154,Z 367.28,A -85,B 0,C 180,E1 -8389.477,E2 -8389.477} C_VEL
LIN {X 0,Y 453.407,Z 359.337,A -85,B 0,C 180,E1 -8392.799,E2 -8392.799} C_VEL
LIN {X 0,Y 453.685,Z 351.847,A -85,B 0,C 180,E1 -8396.041,E2 -8396.041} C_VEL
LIN {X 0,Y 453.983,Z 344.718,A -85,B 0,C 180,E1 -8399.185,E2 -8399.185} C_VEL
LIN {X 0,Y 454.277,Z 337.967,A -85,B 0,C 180,E1 -8402.257,E2 -8402.257} C_VEL
LIN {X 0,Y 454.568,Z 332.187,A -85,B 0,C 180,E1 -8404.973,E2 -8404.973} C_VEL
LIN {X 0,Y 454.312,Z 327.888,A -85,B 0,C 180,E1 -8407.106,E2 -8407.106} C_VEL
LIN {X 0,Y 453.533,Z 322.994,A -85,B 0,C 180,E1 -8409.732,E2 -8409.732} C_VEL
LIN {X 0,Y 453.477,Z 323.003,A -85,B 0,C 180,E1 -8413.247,E2 -8413.247} C_VEL
LIN {X 0,Y 453.456,Z 323.002,A -85,B 0,C 180,E1 -8415.778,E2 -8415.778} C_VEL
LIN {X 0,Y 453.464,Z 322.997,A -85,B 0,C 180,E1 -8419.412,E2 -8419.412} C_VEL
LIN {X 0,Y 453.463,Z 323,A -85,B 0,C 180,E1 -8422.811,E2 -8422.811} C_VEL
LIN {X 0,Y 453.47,Z 323,A -85,B 0,C 180,E1 -8426.087,E2 -8426.087} C_VEL
LIN {X 0,Y 453.465,Z 322.999,A -85,B 0,C 180,E1 -8429.24,E2 -8429.24} C_VEL
LIN {X 0,Y 453.48,Z 322.999,A -85,B 0,C 180,E1 -8432.294,E2 -8432.294} C_VEL
LIN {X 0,Y 453.491,Z 322.994,A -85,B 0,C 180,E1 -8435.264,E2 -8435.264} C_VEL
LIN {X 0,Y 453.471,Z 322.999,A -85,B 0,C 180,E1 -8438.414,E2 -8438.414} C_VEL
LIN {X 0,Y 453.512,Z 322.993,A -85,B 0,C 180,E1 -8441.008,E2 -8441.008} C_VEL
LIN {X 0,Y 453.559,Z 322.988,A -85,B 0,C 180,E1 -8443.879,E2 -8443.879} C_VEL
LIN {X 0,Y 453.553,Z 322.987,A -85,B 0,C 180,E1 -8447.471,E2 -8447.471} C_VEL
LIN {X 0,Y 453.582,Z 322.984,A -85,B 0,C 180,E1 -8451.086,E2 -8451.086} C_VEL
LIN {X 0,Y 453.675,Z 322.974,A -85,B 0,C 180,E1 -8453.775,E2 -8453.775} C_VEL
LIN {X 0,Y 453.755,Z 322.964,A -85,B 0,C 180,E1 -8457.337,E2 -8457.337} C_VEL
LIN {X 0,Y 453.805,Z 322.959,A -85,B 0,C 180,E1 -8460,E2 -8460} C_VEL
LIN {X 0,Y 453.734,Z 322.963,A -85,B 0,C 180,E1 -8462.663,E2 -8462.663} C_VEL
LIN {X 0,Y 453.671,Z 322.974,A -85,B 0,C 180,E1 -8466.225,E2 -8466.225} C_VEL
LIN {X 0,Y 453.582,Z 322.986,A -85,B 0,C 180,E1 -8468.914,E2 -8468.914} C_VEL
LIN {X 0,Y 453.553,Z 322.988,A -85,B 0,C 180,E1 -8472.529,E2 -8472.529} C_VEL
LIN {X 0,Y 453.535,Z 322.987,A -85,B 0,C 180,E1 -8476.196,E2 -8476.196} C_VEL
LIN {X 0,Y 453.511,Z 322.997,A -85,B 0,C 180,E1 -8479.041,E2 -8479.041} C_VEL
LIN {X 0,Y 453.467,Z 322.999,A -85,B 0,C 180,E1 -8481.837,E2 -8481.837} C_VEL
LIN {X 0,Y 453.491,Z 322.997,A -85,B 0,C 180,E1 -8484.736,E2 -8484.736} C_VEL
LIN {X 0,Y 453.466,Z 322.998,A -85,B 0,C 180,E1 -8487.947,E2 -8487.947} C_VEL
LIN {X 0,Y 453.465,Z 323.002,A -85,B 0,C 180,E1 -8490.761,E2 -8490.761} C_VEL
LIN {X 0,Y 453.471,Z 322.997,A -85,B 0,C 180,E1 -8493.913,E2 -8493.913} C_VEL
LIN {X 0,Y 453.447,Z 323.003,A -85,B 0,C 180,E1 -8497.19,E2 -8497.19} C_VEL
LIN {X 0,Y 453.463,Z 323.001,A -85,B 0,C 180,E1 -8500.613,E2 -8500.613} C_VEL
LIN {X 0,Y 453.453,Z 323.001,A -85,B 0,C 180,E1 -8504.223,E2 -8504.223} C_VEL
LIN {X 0,Y 453.458,Z 322.999,A -85,B 0,C 180,E1 -8507.006,E2 -8507.006} C_VEL
LIN {X 0,Y 453.527,Z 322.992,A -85,B 0,C 180,E1 -8510.556,E2 -8510.556} C_VEL
LIN {X 0,Y 453.393,Z 323.01,A -85,B 0,C 180,E1 -8513.913,E2 -8513.913} C_VEL
LIN {X 0,Y 453.395,Z 323.999,A -85,B 0,C 180,E1 -8515.24,E2 -8515.24} C_VEL
LIN {X 0,Y 453.272,Z 327.918,A -85,B 0,C 180,E1 -8518.187,E2 -8518.187} C_VEL
LIN {X 0,Y 453.148,Z 332.129,A -85,B 0,C 180,E1 -8521.264,E2 -8521.264} C_VEL
LIN {X 0,Y 453.021,Z 336.303,A -85,B 0,C 180,E1 -8524.255,E2 -8524.255} C_VEL
LIN {X 0,Y 452.876,Z 340.468,A -85,B 0,C 180,E1 -8527.173,E2 -8527.173} C_VEL
LIN {X 0,Y 452.765,Z 344.692,A -85,B 0,C 180,E1 -8530.033,E2 -8530.033} C_VEL
LIN {X 0,Y 452.688,Z 348.988,A -85,B 0,C 180,E1 -8532.845,E2 -8532.845} C_VEL
LIN {X 0,Y 452.734,Z 351.055,A -85,B 0,C 180,E1 -8534.17,E2 -8534.17} C_VEL
LIN {X 0,Y 455.9,Z 365.983,A -85,B 0,C 180,E1 -8534.751,E2 -8534.751} C_VEL
LIN {X 0,Y 456.435,Z 371.398,A -85,B 0,C 180,E1 -8534.998,E2 -8534.998} C_VEL
LIN {X 0,Y 456.014,Z 383.318,A -85,B 0,C 180,E1 -8535.611,E2 -8535.611} C_VEL
LIN {X 0,Y 455.507,Z 393.869,A -85,B 0,C 180,E1 -8536.318,E2 -8536.318} C_VEL
LIN {X 0,Y 455.075,Z 404.364,A -85,B 0,C 180,E1 -8537.206,E2 -8537.206} C_VEL
LIN {X 0,Y 454.11,Z 409.11,A -85,B 0,C 180,E1 -8537.65,E2 -8537.65} C_VEL
LIN {X 0,Y 450.843,Z 416.483,A -85,B 0,C 180,E1 -8538.391,E2 -8538.391} C_VEL
LIN {X 0,Y 447.643,Z 423.264,A -85,B 0,C 180,E1 -8539.207,E2 -8539.207} C_VEL
LIN {X 0,Y 446.776,Z 427.084,A -85,B 0,C 180,E1 -8539.763,E2 -8539.763} C_VEL
LIN {X 0,Y 446.306,Z 435.067,A -85,B 0,C 180,E1 -8541.169,E2 -8541.169} C_VEL
LIN {X 0,Y 445.886,Z 442.125,A -85,B 0,C 180,E1 -8542.757,E2 -8542.757} C_VEL
LIN {X 0,Y 445.776,Z 446.824,A -85,B 0,C 180,E1 -8544.119,E2 -8544.119} C_VEL
LIN {X 0,Y 445.511,Z 450.427,A -85,B 0,C 180,E1 -8545.477,E2 -8545.477} C_VEL
LIN {X 0,Y 445.527,Z 452.285,A -85,B 0,C 180,E1 -8546.383,E2 -8546.383} C_VEL
LIN {X 0,Y 445.464,Z 453.687,A -85,B 0,C 180,E1 -8547.288,E2 -8547.288} C_VEL
LIN {X 0,Y 445.341,Z 455.3,A -85,B 0,C 180,E1 -8549.096,E2 -8549.096} C_VEL
LIN {X 0,Y 445.342,Z 455.534,A -85,B 0,C 180,E1 -8550,E2 -8550} C_VEL
LIN {X 0,Y 445.341,Z 455.347,A -85,B 0,C 180,E1 -8550.905,E2 -8550.905} C_VEL
LIN {X 0,Y 445.464,Z 453.796,A -85,B 0,C 180,E1 -8552.713,E2 -8552.713} C_VEL
LIN {X 0,Y 445.525,Z 452.441,A -85,B 0,C 180,E1 -8553.618,E2 -8553.618} C_VEL
LIN {X 0,Y 445.542,Z 449.581,A -85,B 0,C 180,E1 -8554.977,E2 -8554.977} C_VEL
LIN {X 0,Y 445.795,Z 445.696,A -85,B 0,C 180,E1 -8556.336,E2 -8556.336} C_VEL
LIN {X 0,Y 445.964,Z 440.689,A -85,B 0,C 180,E1 -8557.698,E2 -8557.698} C_VEL
LIN {X 0,Y 446.36,Z 434.381,A -85,B 0,C 180,E1 -8559.059,E2 -8559.059} C_VEL
LIN {X 0,Y 446.789,Z 426.486,A -85,B 0,C 180,E1 -8560.422,E2 -8560.422} C_VEL
LIN {X 0,Y 447.384,Z 416.662,A -85,B 0,C 180,E1 -8561.784,E2 -8561.784} C_VEL
LIN {X 0,Y 448.064,Z 406.745,A -85,B 0,C 180,E1 -8562.877,E2 -8562.877} C_VEL
LIN {X 0,Y 448.531,Z 395.274,A -85,B 0,C 180,E1 -8563.895,E2 -8563.895} C_VEL
LIN {X 0,Y 449.065,Z 384.964,A -85,B 0,C 180,E1 -8564.617,E2 -8564.617} C_VEL
LIN {X 0,Y 449.593,Z 372.389,A -85,B 0,C 180,E1 -8565.295,E2 -8565.295} C_VEL
LIN {X 0,Y 449.233,Z 368.051,A -85,B 0,C 180,E1 -8565.502,E2 -8565.502} C_VEL
LIN {X 0,Y 446.562,Z 355.376,A -85,B 0,C 180,E1 -8566.033,E2 -8566.033} C_VEL
LIN {X 0,Y 445.583,Z 351.263,A -85,B 0,C 180,E1 -8566.184,E2 -8566.184} C_VEL
LIN {X 0,Y 445.687,Z 346.454,A -85,B 0,C 180,E1 -8569.338,E2 -8569.338} C_VEL
LIN {X 0,Y 445.776,Z 342.192,A -85,B 0,C 180,E1 -8572.233,E2 -8572.233} C_VEL
LIN {X 0,Y 445.906,Z 337.995,A -85,B 0,C 180,E1 -8575.186,E2 -8575.186} C_VEL
LIN {X 0,Y 446.04,Z 333.82,A -85,B 0,C 180,E1 -8578.209,E2 -8578.209} C_VEL
LIN {X 0,Y 446.213,Z 329.587,A -85,B 0,C 180,E1 -8581.316,E2 -8581.316} C_VEL
LIN {X 0,Y 446.352,Z 325.338,A -85,B 0,C 180,E1 -8584.53,E2 -8584.53} C_VEL
LIN {X 0,Y 446.325,Z 323.923,A -85,B 0,C 180,E1 -8585.634,E2 -8585.634} C_VEL
LIN {X 0,Y 446.437,Z 323.877,A -85,B 0,C 180,E1 -8589.027,E2 -8589.027} C_VEL
LIN {X 0,Y 446.434,Z 323.875,A -85,B 0,C 180,E1 -8592.277,E2 -8592.277} C_VEL
LIN {X 0,Y 446.449,Z 323.872,A -85,B 0,C 180,E1 -8595.104,E2 -8595.104} C_VEL
LIN {X 0,Y 446.398,Z 323.878,A -85,B 0,C 180,E1 -8598.605,E2 -8598.605} C_VEL
LIN {X 0,Y 446.41,Z 323.879,A -85,B 0,C 180,E1 -8601.921,E2 -8601.921} C_VEL
LIN {X 0,Y 446.428,Z 323.879,A -85,B 0,C 180,E1 -8605.477,E2 -8605.477} C_VEL
LIN {X 0,Y 446.411,Z 323.877,A -85,B 0,C 180,E1 -8608.699,E2 -8608.699} C_VEL
LIN {X 0,Y 446.422,Z 323.876,A -85,B 0,C 180,E1 -8611.835,E2 -8611.835} C_VEL
LIN {X 0,Y 446.428,Z 323.878,A -85,B 0,C 180,E1 -8614.846,E2 -8614.846} C_VEL
LIN {X 0,Y 446.444,Z 323.874,A -85,B 0,C 180,E1 -8618.245,E2 -8618.245} C_VEL
LIN {X 0,Y 446.452,Z 323.871,A -85,B 0,C 180,E1 -8621.649,E2 -8621.649} C_VEL
LIN {X 0,Y 446.501,Z 323.867,A -85,B 0,C 180,E1 -8624.479,E2 -8624.479} C_VEL
LIN {X 0,Y 446.513,Z 323.866,A -85,B 0,C 180,E1 -8628.193,E2 -8628.193} C_VEL
LIN {X 0,Y 446.596,Z 323.855,A -85,B 0,C 180,E1 -8631.858,E2 -8631.858} C_VEL
LIN {X 0,Y 446.643,Z 323.852,A -85,B 0,C 180,E1 -8634.583,E2 -8634.583} C_VEL
LIN {X 0,Y 446.657,Z 323.849,A -85,B 0,C 180,E1 -8638.197,E2 -8638.197} C_VEL
LIN {X 0,Y 446.779,Z 323.833,A -85,B 0,C 180,E1 -8640,E2 -8640} C_VEL
LIN {X 0,Y 446.685,Z 323.844,A -85,B 0,C 180,E1 -8642.705,E2 -8642.705} C_VEL
LIN {X 0,Y 446.643,Z 323.851,A -85,B 0,C 180,E1 -8646.324,E2 -8646.324} C_VEL
LIN {X 0,Y 446.534,Z 323.861,A -85,B 0,C 180,E1 -8649.055,E2 -8649.055} C_VEL
LIN {X 0,Y 446.517,Z 323.863,A -85,B 0,C 180,E1 -8652.73,E2 -8652.73} C_VEL
LIN {X 0,Y 446.485,Z 323.869,A -85,B 0,C 180,E1 -8656.459,E2 -8656.459} C_VEL
LIN {X 0,Y 446.466,Z 323.872,A -85,B 0,C 180,E1 -8659.303,E2 -8659.303} C_VEL
LIN {X 0,Y 446.415,Z 323.879,A -85,B 0,C 180,E1 -8662.2,E2 -8662.2} C_VEL
LIN {X 0,Y 446.437,Z 323.874,A -85,B 0,C 180,E1 -8665.154,E2 -8665.154} C_VEL
LIN {X 0,Y 446.434,Z 323.874,A -85,B 0,C 180,E1 -8668.182,E2 -8668.182} C_VEL
LIN {X 0,Y 446.411,Z 323.88,A -85,B 0,C 180,E1 -8671.301,E2 -8671.301} C_VEL
LIN {X 0,Y 446.428,Z 323.875,A -85,B 0,C 180,E1 -8674.523,E2 -8674.523} C_VEL
LIN {X 0,Y 446.424,Z 323.875,A -85,B 0,C 180,E1 -8678.081,E2 -8678.081} C_VEL
LIN {X 0,Y 446.397,Z 323.881,A -85,B 0,C 180,E1 -8681.395,E2 -8681.395} C_VEL
LIN {X 0,Y 446.449,Z 323.875,A -85,B 0,C 180,E1 -8685.104,E2 -8685.104} C_VEL
LIN {X 0,Y 446.428,Z 323.877,A -85,B 0,C 180,E1 -8688.609,E2 -8688.609} C_VEL
LIN {X 0,Y 446.499,Z 324.055,A -85,B 0,C 180,E1 -8690.172,E2 -8690.172} C_VEL
LIN {X 0,Y 447.419,Z 329.798,A -85,B 0,C 180,E1 -8693.236,E2 -8693.236} C_VEL
LIN {X 0,Y 447.609,Z 332.773,A -85,B 0,C 180,E1 -8694.732,E2 -8694.732} C_VEL
LIN {X 0,Y 447.252,Z 339.713,A -85,B 0,C 180,E1 -8698.054,E2 -8698.054} C_VEL
LIN {X 0,Y 446.968,Z 345.722,A -85,B 0,C 180,E1 -8700.828,E2 -8700.828} C_VEL
LIN {X 0,Y 446.657,Z 352.489,A -85,B 0,C 180,E1 -8703.86,E2 -8703.86} C_VEL
LIN {X 0,Y 446.334,Z 360.383,A -85,B 0,C 180,E1 -8707.308,E2 -8707.308} C_VEL
LIN {X 0,Y 446.083,Z 368.255,A -85,B 0,C 180,E1 -8710.679,E2 -8710.679} C_VEL
LIN {X 0,Y 445.876,Z 375.721,A -85,B 0,C 180,E1 -8713.844,E2 -8713.844} C_VEL
LIN {X 0,Y 448.373,Z 389.912,A -85,B 0,C 180,E1 -8714.345,E2 -8714.345} C_VEL
LIN {X 0,Y 449.418,Z 397.67,A -85,B 0,C 180,E1 -8714.699,E2 -8714.699} C_VEL
LIN {X 0,Y 448.963,Z 408.708,A -85,B 0,C 180,E1 -8715.263,E2 -8715.263} C_VEL
LIN {X 0,Y 448.398,Z 420.57,A -85,B 0,C 180,E1 -8716.055,E2 -8716.055} C_VEL
LIN {X 0,Y 447.81,Z 431.497,A -85,B 0,C 180,E1 -8716.99,E2 -8716.99} C_VEL
LIN {X 0,Y 447.289,Z 440.92,A -85,B 0,C 180,E1 -8717.984,E2 -8717.984} C_VEL
LIN {X 0,Y 446.72,Z 449.772,A -85,B 0,C 180,E1 -8719.118,E2 -8719.118} C_VEL
LIN {X 0,Y 446.282,Z 458.409,A -85,B 0,C 180,E1 -8720.482,E2 -8720.482} C_VEL
LIN {X 0,Y 445.884,Z 465.311,A -85,B 0,C 180,E1 -8721.844,E2 -8721.844} C_VEL
LIN {X 0,Y 445.658,Z 470.847,A -85,B 0,C 180,E1 -8723.208,E2 -8723.208} C_VEL
LIN {X 0,Y 445.541,Z 475.187,A -85,B 0,C 180,E1 -8724.569,E2 -8724.569} C_VEL
LIN {X 0,Y 445.427,Z 477.483,A -85,B 0,C 180,E1 -8725.475,E2 -8725.475} C_VEL
LIN {X 0,Y 445.387,Z 479.346,A -85,B 0,C 180,E1 -8726.381,E2 -8726.381} C_VEL
LIN {X 0,Y 445.422,Z 480.746,A -85,B 0,C 180,E1 -8727.287,E2 -8727.287} C_VEL
LIN {X 0,Y 445.315,Z 482.349,A -85,B 0,C 180,E1 -8729.095,E2 -8729.095} C_VEL
LIN {X 0,Y 445.292,Z 482.565,A -85,B 0,C 180,E1 -8730,E2 -8730} C_VEL
LIN {X 0,Y 445.315,Z 482.35,A -85,B 0,C 180,E1 -8730.904,E2 -8730.904} C_VEL
LIN {X 0,Y 445.422,Z 480.75,A -85,B 0,C 180,E1 -8732.713,E2 -8732.713} C_VEL
LIN {X 0,Y 445.387,Z 479.352,A -85,B 0,C 180,E1 -8733.618,E2 -8733.618} C_VEL
LIN {X 0,Y 445.5,Z 476.416,A -85,B 0,C 180,E1 -8734.977,E2 -8734.977} C_VEL
LIN {X 0,Y 445.584,Z 472.076,A -85,B 0,C 180,E1 -8736.448,E2 -8736.448} C_VEL
LIN {X 0,Y 445.807,Z 466.328,A -85,B 0,C 180,E1 -8737.928,E2 -8737.928} C_VEL
LIN {X 0,Y 446.193,Z 459.651,A -85,B 0,C 180,E1 -8739.29,E2 -8739.29} C_VEL
LIN {X 0,Y 446.643,Z 451.366,A -85,B 0,C 180,E1 -8740.654,E2 -8740.654} C_VEL
LIN {X 0,Y 447.185,Z 442.878,A -85,B 0,C 180,E1 -8741.788,E2 -8741.788} C_VEL
LIN {X 0,Y 447.744,Z 433.141,A -85,B 0,C 180,E1 -8742.851,E2 -8742.851} C_VEL
LIN {X 0,Y 448.284,Z 422.012,A -85,B 0,C 180,E1 -8743.832,E2 -8743.832} C_VEL
LIN {X 0,Y 448.871,Z 410.64,A -85,B 0,C 180,E1 -8744.623,E2 -8744.623} C_VEL
LIN {X 0,Y 449.378,Z 398.981,A -85,B 0,C 180,E1 -8745.244,E2 -8745.244} C_VEL
LIN {X 0,Y 448.366,Z 389.878,A -85,B 0,C 180,E1 -8745.656,E2 -8745.656} C_VEL
LIN {X 0,Y 446.02,Z 376.988,A -85,B 0,C 180,E1 -8746.118,E2 -8746.118} C_VEL
LIN {X 0,Y 445.882,Z 375.714,A -85,B 0,C 180,E1 -8746.158,E2 -8746.158} C_VEL
LIN {X 0,Y 446.12,Z 367.13,A -85,B 0,C 180,E1 -8749.797,E2 -8749.797} C_VEL
LIN {X 0,Y 446.381,Z 359.245,A -85,B 0,C 180,E1 -8753.178,E2 -8753.178} C_VEL
LIN {X 0,Y 446.687,Z 351.34,A -85,B 0,C 180,E1 -8756.648,E2 -8756.648} C_VEL
LIN {X 0,Y 447.02,Z 344.632,A -85,B 0,C 180,E1 -8759.665,E2 -8759.665} C_VEL
LIN {X 0,Y 447.267,Z 338.974,A -85,B 0,C 180,E1 -8762.292,E2 -8762.292} C_VEL
LIN {X 0,Y 447.609,Z 332.754,A -85,B 0,C 180,E1 -8765.268,E2 -8765.268} C_VEL
LIN {X 0,Y 447.418,Z 329.791,A -85,B 0,C 180,E1 -8766.764,E2 -8766.764} C_VEL
LIN {X 0,Y 446.496,Z 323.871,A -85,B 0,C 180,E1 -8769.92,E2 -8769.92} C_VEL
LIN {X 0,Y 446.442,Z 323.881,A -85,B 0,C 180,E1 -8773.602,E2 -8773.602} C_VEL
LIN {X 0,Y 446.387,Z 323.881,A -85,B 0,C 180,E1 -8776.403,E2 -8776.403} C_VEL
LIN {X 0,Y 446.393,Z 323.877,A -85,B 0,C 180,E1 -8779.796,E2 -8779.796} C_VEL
LIN {X 0,Y 446.418,Z 323.877,A -85,B 0,C 180,E1 -8782.122,E2 -8782.122} C_VEL
LIN {X 0,Y 446.423,Z 323.876,A -85,B 0,C 180,E1 -8785.476,E2 -8785.476} C_VEL
LIN {X 0,Y 446.406,Z 323.881,A -85,B 0,C 180,E1 -8788.699,E2 -8788.699} C_VEL
LIN {X 0,Y 446.437,Z 323.873,A -85,B 0,C 180,E1 -8791.83,E2 -8791.83} C_VEL
LIN {X 0,Y 446.433,Z 323.874,A -85,B 0,C 180,E1 -8794.846,E2 -8794.846} C_VEL
LIN {X 0,Y 446.439,Z 323.876,A -85,B 0,C 180,E1 -8798.244,E2 -8798.244} C_VEL
LIN {X 0,Y 446.447,Z 323.875,A -85,B 0,C 180,E1 -8801.649,E2 -8801.649} C_VEL
LIN {X 0,Y 446.495,Z 323.869,A -85,B 0,C 180,E1 -8804.479,E2 -8804.479} C_VEL
LIN {X 0,Y 446.507,Z 323.867,A -85,B 0,C 180,E1 -8808.193,E2 -8808.193} C_VEL
LIN {X 0,Y 446.59,Z 323.858,A -85,B 0,C 180,E1 -8811.858,E2 -8811.858} C_VEL
LIN {X 0,Y 446.643,Z 323.849,A -85,B 0,C 180,E1 -8814.583,E2 -8814.583} C_VEL
LIN {X 0,Y 446.699,Z 323.843,A -85,B 0,C 180,E1 -8817.295,E2 -8817.295} C_VEL
LIN {X 0,Y 446.775,Z 323.834,A -85,B 0,C 180,E1 -8820,E2 -8820} C_VEL
LIN {X 0,Y 446.682,Z 323.841,A -85,B 0,C 180,E1 -8822.706,E2 -8822.706} C_VEL
LIN {X 0,Y 446.64,Z 323.849,A -85,B 0,C 180,E1 -8826.324,E2 -8826.324} C_VEL
LIN {X 0,Y 446.528,Z 323.866,A -85,B 0,C 180,E1 -8829.056,E2 -8829.056} C_VEL
LIN {X 0,Y 446.511,Z 323.866,A -85,B 0,C 180,E1 -8832.73,E2 -8832.73} C_VEL
LIN {X 0,Y 446.48,Z 323.866,A -85,B 0,C 180,E1 -8836.46,E2 -8836.46} C_VEL
LIN {X 0,Y 446.46,Z 323.873,A -85,B 0,C 180,E1 -8839.304,E2 -8839.304} C_VEL
LIN {X 0,Y 446.409,Z 323.878,A -85,B 0,C 180,E1 -8842.2,E2 -8842.2} C_VEL
LIN {X 0,Y 446.433,Z 323.877,A -85,B 0,C 180,E1 -8845.154,E2 -8845.154} C_VEL
LIN {X 0,Y 446.429,Z 323.875,A -85,B 0,C 180,E1 -8848.183,E2 -8848.183} C_VEL
LIN {X 0,Y 446.406,Z 323.878,A -85,B 0,C 180,E1 -8851.301,E2 -8851.301} C_VEL
LIN {X 0,Y 446.424,Z 323.879,A -85,B 0,C 180,E1 -8854.524,E2 -8854.524} C_VEL
LIN {X 0,Y 446.406,Z 323.879,A -85,B 0,C 180,E1 -8858.08,E2 -8858.08} C_VEL
LIN {X 0,Y 446.398,Z 323.878,A -85,B 0,C 180,E1 -8861.395,E2 -8861.395} C_VEL
LIN {X 0,Y 446.445,Z 323.872,A -85,B 0,C 180,E1 -8865.105,E2 -8865.105} C_VEL
LIN {X 0,Y 446.432,Z 323.876,A -85,B 0,C 180,E1 -8868.611,E2 -8868.611} C_VEL
LIN {X 0,Y 446.468,Z 323.871,A -85,B 0,C 180,E1 -8870.977,E2 -8870.977} C_VEL
LIN {X 0,Y 446.311,Z 323.893,A -85,B 0,C 180,E1 -8874.365,E2 -8874.365} C_VEL
LIN {X 0,Y 446.327,Z 326.646,A -85,B 0,C 180,E1 -8876.57,E2 -8876.57} C_VEL
LIN {X 0,Y 446.162,Z 331.275,A -85,B 0,C 180,E1 -8880.04,E2 -8880.04} C_VEL
LIN {X 0,Y 446.003,Z 335.07,A -85,B 0,C 180,E1 -8882.809,E2 -8882.809} C_VEL
LIN {X 0,Y 445.889,Z 339.643,A -85,B 0,C 180,E1 -8886.091,E2 -8886.091} C_VEL
LIN {X 0,Y 445.726,Z 344.875,A -85,B 0,C 180,E1 -8889.704,E2 -8889.704} C_VEL
LIN {X 0,Y 445.638,Z 349.189,A -85,B 0,C 180,E1 -8892.565,E2 -8892.565} C_VEL
LIN {X 0,Y 445.648,Z 351.311,A -85,B 0,C 180,E1 -8893.922,E2 -8893.922} C_VEL
LIN {X 0,Y 448.502,Z 364.257,A -85,B 0,C 180,E1 -8894.417,E2 -8894.417} C_VEL
LIN {X 0,Y 449.603,Z 371.623,A -85,B 0,C 180,E1 -8894.764,E2 -8894.764} C_VEL
LIN {X 0,Y 449.145,Z 383.541,A -85,B 0,C 180,E1 -8895.386,E2 -8895.386} C_VEL
LIN {X 0,Y 448.546,Z 395.302,A -85,B 0,C 180,E1 -8896.2,E2 -8896.2} C_VEL
LIN {X 0,Y 448.026,Z 406.744,A -85,B 0,C 180,E1 -8897.214,E2 -8897.214} C_VEL
LIN {X 0,Y 447.458,Z 415.917,A -85,B 0,C 180,E1 -8898.219,E2 -8898.219} C_VEL
LIN {X 0,Y 446.962,Z 424.415,A -85,B 0,C 180,E1 -8899.354,E2 -8899.354} C_VEL
LIN {X 0,Y 446.776,Z 427.084,A -85,B 0,C 180,E1 -8899.763,E2 -8899.763} C_VEL
LIN {X 0,Y 445.903,Z 430.761,A -85,B 0,C 180,E1 -8900.346,E2 -8900.346} C_VEL
LIN {X 0,Y 442.695,Z 436.289,A -85,B 0,C 180,E1 -8901.325,E2 -8901.325} C_VEL
LIN {X 0,Y 439.543,Z 441.235,A -85,B 0,C 180,E1 -8902.37,E2 -8902.37} C_VEL
LIN {X 0,Y 438.768,Z 443.857,A -85,B 0,C 180,E1 -8903.052,E2 -8903.052} C_VEL
LIN {X 0,Y 438.606,Z 448.356,A -85,B 0,C 180,E1 -8904.484,E2 -8904.484} C_VEL
LIN {X 0,Y 438.433,Z 450.644,A -85,B 0,C 180,E1 -8905.403,E2 -8905.403} C_VEL
LIN {X 0,Y 438.431,Z 452.501,A -85,B 0,C 180,E1 -8906.324,E2 -8906.324} C_VEL
LIN {X 0,Y 438.395,Z 453.902,A -85,B 0,C 180,E1 -8907.244,E2 -8907.244} C_VEL
LIN {X 0,Y 438.255,Z 455.515,A -85,B 0,C 180,E1 -8909.082,E2 -8909.082} C_VEL
LIN {X 0,Y 438.254,Z 455.749,A -85,B 0,C 180,E1 -8910,E2 -8910} C_VEL
LIN {X 0,Y 438.255,Z 455.562,A -85,B 0,C 180,E1 -8910.919,E2 -8910.919} C_VEL
LIN {X 0,Y 438.395,Z 454.01,A -85,B 0,C 180,E1 -8912.757,E2 -8912.757} C_VEL
LIN {X 0,Y 438.429,Z 452.656,A -85,B 0,C 180,E1 -8913.677,E2 -8913.677} C_VEL
LIN {X 0,Y 438.484,Z 449.795,A -85,B 0,C 180,E1 -8915.058,E2 -8915.058} C_VEL
LIN {X 0,Y 438.71,Z 445.911,A -85,B 0,C 180,E1 -8916.439,E2 -8916.439} C_VEL
LIN {X 0,Y 438.912,Z 440.903,A -85,B 0,C 180,E1 -8917.823,E2 -8917.823} C_VEL
LIN {X 0,Y 439.329,Z 434.595,A -85,B 0,C 180,E1 -8919.205,E2 -8919.205} C_VEL
LIN {X 0,Y 439.816,Z 426.698,A -85,B 0,C 180,E1 -8920.589,E2 -8920.589} C_VEL
LIN {X 0,Y 440.437,Z 416.874,A -85,B 0,C 180,E1 -8921.973,E2 -8921.973} C_VEL
LIN {X 0,Y 441.135,Z 407.091,A -85,B 0,C 180,E1 -8923.069,E2 -8923.069} C_VEL
LIN {X 0,Y 441.61,Z 396.35,A -85,B 0,C 180,E1 -8924.046,E2 -8924.046} C_VEL
LIN {X 0,Y 442.219,Z 385.172,A -85,B 0,C 180,E1 -8924.849,E2 -8924.849} C_VEL
LIN {X 0,Y 442.758,Z 372.594,A -85,B 0,C 180,E1 -8925.537,E2 -8925.537} C_VEL
LIN {X 0,Y 441.4,Z 363.966,A -85,B 0,C 180,E1 -8925.954,E2 -8925.954} C_VEL
LIN {X 0,Y 438.513,Z 351.47,A -85,B 0,C 180,E1 -8926.454,E2 -8926.454} C_VEL
LIN {X 0,Y 438.633,Z 346.642,A -85,B 0,C 180,E1 -8929.662,E2 -8929.662} C_VEL
LIN {X 0,Y 438.713,Z 342.367,A -85,B 0,C 180,E1 -8932.611,E2 -8932.611} C_VEL
LIN {X 0,Y 438.861,Z 338.154,A -85,B 0,C 180,E1 -8935.619,E2 -8935.619} C_VEL
LIN {X 0,Y 439.014,Z 333.963,A -85,B 0,C 180,E1 -8938.702,E2 -8938.702} C_VEL
LIN {X 0,Y 439.194,Z 329.715,A -85,B 0,C 180,E1 -8941.875,E2 -8941.875} C_VEL
LIN {X 0,Y 439.28,Z 326.872,A -85,B 0,C 180,E1 -8944.053,E2 -8944.053} C_VEL
LIN {X 0,Y 439.315,Z 325.249,A -85,B 0,C 180,E1 -8945.325,E2 -8945.325} C_VEL
LIN {X 0,Y 439.334,Z 324.765,A -85,B 0,C 180,E1 -8946.884,E2 -8946.884} C_VEL
LIN {X 0,Y 439.402,Z 324.753,A -85,B 0,C 180,E1 -8949.849,E2 -8949.849} C_VEL
LIN {X 0,Y 439.381,Z 324.752,A -85,B 0,C 180,E1 -8952.626,E2 -8952.626} C_VEL
LIN {X 0,Y 439.396,Z 324.752,A -85,B 0,C 180,E1 -8955.27,E2 -8955.27} C_VEL
LIN {X 0,Y 439.351,Z 324.758,A -85,B 0,C 180,E1 -8959.016,E2 -8959.016} C_VEL
LIN {X 0,Y 439.345,Z 324.758,A -85,B 0,C 180,E1 -8962.564,E2 -8962.564} C_VEL
LIN {X 0,Y 439.399,Z 324.752,A -85,B 0,C 180,E1 -8964.844,E2 -8964.844} C_VEL
LIN {X 0,Y 439.369,Z 324.753,A -85,B 0,C 180,E1 -8968.139,E2 -8968.139} C_VEL
LIN {X 0,Y 439.397,Z 324.751,A -85,B 0,C 180,E1 -8971.606,E2 -8971.606} C_VEL
LIN {X 0,Y 439.368,Z 324.755,A -85,B 0,C 180,E1 -8974.413,E2 -8974.413} C_VEL
LIN {X 0,Y 439.359,Z 324.758,A -85,B 0,C 180,E1 -8977.424,E2 -8977.424} C_VEL
LIN {X 0,Y 439.438,Z 324.747,A -85,B 0,C 180,E1 -8980.663,E2 -8980.663} C_VEL
LIN {X 0,Y 439.457,Z 324.742,A -85,B 0,C 180,E1 -8984.224,E2 -8984.224} C_VEL
LIN {X 0,Y 439.479,Z 324.741,A -85,B 0,C 180,E1 -8988.001,E2 -8988.001} C_VEL
LIN {X 0,Y 439.544,Z 324.733,A -85,B 0,C 180,E1 -8991.726,E2 -8991.726} C_VEL
LIN {X 0,Y 439.618,Z 324.726,A -85,B 0,C 180,E1 -8994.496,E2 -8994.496} C_VEL
LIN {X 0,Y 439.628,Z 324.724,A -85,B 0,C 180,E1 -8998.168,E2 -8998.168} C_VEL
LIN {X 0,Y 439.748,Z 324.709,A -85,B 0,C 180,E1 -9000,E2 -9000} C_VEL
LIN {X 0,Y 439.635,Z 324.723,A -85,B 0,C 180,E1 -9002.749,E2 -9002.749} C_VEL
LIN {X 0,Y 439.614,Z 324.727,A -85,B 0,C 180,E1 -9006.425,E2 -9006.425} C_VEL
LIN {X 0,Y 439.496,Z 324.738,A -85,B 0,C 180,E1 -9009.202,E2 -9009.202} C_VEL
LIN {X 0,Y 439.46,Z 324.741,A -85,B 0,C 180,E1 -9012.938,E2 -9012.938} C_VEL
LIN {X 0,Y 439.443,Z 324.746,A -85,B 0,C 180,E1 -9016.349,E2 -9016.349} C_VEL
LIN {X 0,Y 439.399,Z 324.753,A -85,B 0,C 180,E1 -9019.626,E2 -9019.626} C_VEL
LIN {X 0,Y 439.361,Z 324.755,A -85,B 0,C 180,E1 -9022.576,E2 -9022.576} C_VEL
LIN {X 0,Y 439.374,Z 324.757,A -85,B 0,C 180,E1 -9025.587,E2 -9025.587} C_VEL
LIN {X 0,Y 439.386,Z 324.751,A -85,B 0,C 180,E1 -9028.676,E2 -9028.676} C_VEL
LIN {X 0,Y 439.366,Z 324.756,A -85,B 0,C 180,E1 -9032.031,E2 -9032.031} C_VEL
LIN {X 0,Y 439.393,Z 324.753,A -85,B 0,C 180,E1 -9035.341,E2 -9035.341} C_VEL
LIN {X 0,Y 439.365,Z 324.754,A -85,B 0,C 180,E1 -9038.597,E2 -9038.597} C_VEL
LIN {X 0,Y 439.346,Z 324.756,A -85,B 0,C 180,E1 -9042.21,E2 -9042.21} C_VEL
LIN {X 0,Y 439.397,Z 324.753,A -85,B 0,C 180,E1 -9045.271,E2 -9045.271} C_VEL
LIN {X 0,Y 439.388,Z 324.754,A -85,B 0,C 180,E1 -9048.744,E2 -9048.744} C_VEL
LIN {X 0,Y 439.462,Z 324.929,A -85,B 0,C 180,E1 -9049.923,E2 -9049.923} C_VEL
LIN {X 0,Y 440.345,Z 330.473,A -85,B 0,C 180,E1 -9052.941,E2 -9052.941} C_VEL
LIN {X 0,Y 440.573,Z 334.391,A -85,B 0,C 180,E1 -9054.952,E2 -9054.952} C_VEL
LIN {X 0,Y 440.21,Z 341.104,A -85,B 0,C 180,E1 -9058.207,E2 -9058.207} C_VEL
LIN {X 0,Y 439.847,Z 348.15,A -85,B 0,C 180,E1 -9061.499,E2 -9061.499} C_VEL
LIN {X 0,Y 439.532,Z 354.604,A -85,B 0,C 180,E1 -9064.423,E2 -9064.423} C_VEL
LIN {X 0,Y 439.265,Z 361.34,A -85,B 0,C 180,E1 -9067.419,E2 -9067.419} C_VEL
LIN {X 0,Y 439.007,Z 369.135,A -85,B 0,C 180,E1 -9070.826,E2 -9070.826} C_VEL
LIN {X 0,Y 438.804,Z 375.464,A -85,B 0,C 180,E1 -9073.562,E2 -9073.562} C_VEL
LIN {X 0,Y 441.553,Z 391.245,A -85,B 0,C 180,E1 -9074.157,E2 -9074.157} C_VEL
LIN {X 0,Y 442.508,Z 398.757,A -85,B 0,C 180,E1 -9074.513,E2 -9074.513} C_VEL
LIN {X 0,Y 441.971,Z 410.413,A -85,B 0,C 180,E1 -9075.143,E2 -9075.143} C_VEL
LIN {X 0,Y 441.418,Z 421.784,A -85,B 0,C 180,E1 -9075.948,E2 -9075.948} C_VEL
LIN {X 0,Y 440.748,Z 433.07,A -85,B 0,C 180,E1 -9076.956,E2 -9076.956} C_VEL
LIN {X 0,Y 440.192,Z 442.654,A -85,B 0,C 180,E1 -9078.021,E2 -9078.021} C_VEL
LIN {X 0,Y 439.627,Z 451.144,A -85,B 0,C 180,E1 -9079.173,E2 -9079.173} C_VEL
LIN {X 0,Y 439.166,Z 459.43,A -85,B 0,C 180,E1 -9080.559,E2 -9080.559} C_VEL
LIN {X 0,Y 438.753,Z 466.108,A -85,B 0,C 180,E1 -9081.943,E2 -9081.943} C_VEL
LIN {X 0,Y 438.526,Z 472.224,A -85,B 0,C 180,E1 -9083.558,E2 -9083.558} C_VEL
LIN {X 0,Y 438.415,Z 476.197,A -85,B 0,C 180,E1 -9084.941,E2 -9084.941} C_VEL
LIN {X 0,Y 438.289,Z 479.131,A -85,B 0,C 180,E1 -9086.322,E2 -9086.322} C_VEL
LIN {X 0,Y 438.332,Z 480.53,A -85,B 0,C 180,E1 -9087.243,E2 -9087.243} C_VEL
LIN {X 0,Y 438.23,Z 482.134,A -85,B 0,C 180,E1 -9089.081,E2 -9089.081} C_VEL
LIN {X 0,Y 438.205,Z 482.35,A -85,B 0,C 180,E1 -9090,E2 -9090} C_VEL
LIN {X 0,Y 438.23,Z 482.135,A -85,B 0,C 180,E1 -9090.918,E2 -9090.918} C_VEL
LIN {X 0,Y 438.332,Z 480.534,A -85,B 0,C 180,E1 -9092.757,E2 -9092.757} C_VEL
LIN {X 0,Y 438.289,Z 479.136,A -85,B 0,C 180,E1 -9093.677,E2 -9093.677} C_VEL
LIN {X 0,Y 438.414,Z 476.2,A -85,B 0,C 180,E1 -9095.058,E2 -9095.058} C_VEL
LIN {X 0,Y 438.505,Z 472.224,A -85,B 0,C 180,E1 -9096.441,E2 -9096.441} C_VEL
LIN {X 0,Y 438.754,Z 466.111,A -85,B 0,C 180,E1 -9098.056,E2 -9098.056} C_VEL
LIN {X 0,Y 439.165,Z 459.435,A -85,B 0,C 180,E1 -9099.44,E2 -9099.44} C_VEL
LIN {X 0,Y 439.628,Z 451.149,A -85,B 0,C 180,E1 -9100.826,E2 -9100.826} C_VEL
LIN {X 0,Y 440.212,Z 442.662,A -85,B 0,C 180,E1 -9101.978,E2 -9101.978} C_VEL
LIN {X 0,Y 440.781,Z 433.111,A -85,B 0,C 180,E1 -9103.039,E2 -9103.039} C_VEL
LIN {X 0,Y 441.382,Z 421.796,A -85,B 0,C 180,E1 -9104.052,E2 -9104.052} C_VEL
LIN {X 0,Y 441.98,Z 410.424,A -85,B 0,C 180,E1 -9104.856,E2 -9104.856} C_VEL
LIN {X 0,Y 442.539,Z 398.766,A -85,B 0,C 180,E1 -9105.485,E2 -9105.485} C_VEL
LIN {X 0,Y 440.694,Z 386.083,A -85,B 0,C 180,E1 -9106.059,E2 -9106.059} C_VEL
LIN {X 0,Y 438.803,Z 375.47,A -85,B 0,C 180,E1 -9106.435,E2 -9106.435} C_VEL
LIN {X 0,Y 439.024,Z 368.059,A -85,B 0,C 180,E1 -9109.643,E2 -9109.643} C_VEL
LIN {X 0,Y 439.307,Z 360.231,A -85,B 0,C 180,E1 -9113.075,E2 -9113.075} C_VEL
LIN {X 0,Y 439.652,Z 352.345,A -85,B 0,C 180,E1 -9116.588,E2 -9116.588} C_VEL
LIN {X 0,Y 439.997,Z 345.587,A -85,B 0,C 180,E1 -9119.679,E2 -9119.679} C_VEL
LIN {X 0,Y 440.308,Z 338.858,A -85,B 0,C 180,E1 -9122.866,E2 -9122.866} C_VEL
LIN {X 0,Y 440.608,Z 333.35,A -85,B 0,C 180,E1 -9125.562,E2 -9125.562} C_VEL
LIN {X 0,Y 440.1,Z 328.864,A -85,B 0,C 180,E1 -9127.911,E2 -9127.911} C_VEL
LIN {X 0,Y 439.466,Z 324.748,A -85,B 0,C 180,E1 -9130.227,E2 -9130.227} C_VEL
LIN {X 0,Y 439.389,Z 324.76,A -85,B 0,C 180,E1 -9133.453,E2 -9133.453} C_VEL
LIN {X 0,Y 439.337,Z 324.759,A -85,B 0,C 180,E1 -9136.539,E2 -9136.539} C_VEL
LIN {X 0,Y 439.35,Z 324.759,A -85,B 0,C 180,E1 -9139.016,E2 -9139.016} C_VEL
LIN {X 0,Y 439.366,Z 324.754,A -85,B 0,C 180,E1 -9141.607,E2 -9141.607} C_VEL
LIN {X 0,Y 439.394,Z 324.753,A -85,B 0,C 180,E1 -9144.843,E2 -9144.843} C_VEL
LIN {X 0,Y 439.364,Z 324.757,A -85,B 0,C 180,E1 -9148.139,E2 -9148.139} C_VEL
LIN {X 0,Y 439.391,Z 324.751,A -85,B 0,C 180,E1 -9151.605,E2 -9151.605} C_VEL
LIN {X 0,Y 439.37,Z 324.758,A -85,B 0,C 180,E1 -9154.413,E2 -9154.413} C_VEL
LIN {X 0,Y 439.355,Z 324.756,A -85,B 0,C 180,E1 -9157.424,E2 -9157.424} C_VEL
LIN {X 0,Y 439.432,Z 324.749,A -85,B 0,C 180,E1 -9160.662,E2 -9160.662} C_VEL
LIN {X 0,Y 439.451,Z 324.747,A -85,B 0,C 180,E1 -9164.224,E2 -9164.224} C_VEL
LIN {X 0,Y 439.473,Z 324.746,A -85,B 0,C 180,E1 -9168.001,E2 -9168.001} C_VEL
LIN {X 0,Y 439.538,Z 324.737,A -85,B 0,C 180,E1 -9171.726,E2 -9171.726} C_VEL
LIN {X 0,Y 439.618,Z 324.724,A -85,B 0,C 180,E1 -9174.496,E2 -9174.496} C_VEL
LIN {X 0,Y 439.623,Z 324.725,A -85,B 0,C 180,E1 -9178.168,E2 -9178.168} C_VEL
LIN {X 0,Y 439.744,Z 324.71,A -85,B 0,C 180,E1 -9180,E2 -9180} C_VEL
LIN {X 0,Y 439.631,Z 324.72,A -85,B 0,C 180,E1 -9182.749,E2 -9182.749} C_VEL
LIN {X 0,Y 439.611,Z 324.724,A -85,B 0,C 180,E1 -9186.425,E2 -9186.425} C_VEL
LIN {X 0,Y 439.49,Z 324.742,A -85,B 0,C 180,E1 -9189.202,E2 -9189.202} C_VEL
LIN {X 0,Y 439.455,Z 324.745,A -85,B 0,C 180,E1 -9192.938,E2 -9192.938} C_VEL
LIN {X 0,Y 439.438,Z 324.743,A -85,B 0,C 180,E1 -9196.349,E2 -9196.349} C_VEL
LIN {X 0,Y 439.393,Z 324.752,A -85,B 0,C 180,E1 -9199.627,E2 -9199.627} C_VEL
LIN {X 0,Y 439.355,Z 324.758,A -85,B 0,C 180,E1 -9202.576,E2 -9202.576} C_VEL
LIN {X 0,Y 439.37,Z 324.755,A -85,B 0,C 180,E1 -9205.587,E2 -9205.587} C_VEL
LIN {X 0,Y 439.381,Z 324.754,A -85,B 0,C 180,E1 -9208.676,E2 -9208.676} C_VEL
LIN {X 0,Y 439.361,Z 324.754,A -85,B 0,C 180,E1 -9212.031,E2 -9212.031} C_VEL
LIN {X 0,Y 439.389,Z 324.753,A -85,B 0,C 180,E1 -9215.342,E2 -9215.342} C_VEL
LIN {X 0,Y 439.356,Z 324.758,A -85,B 0,C 180,E1 -9218.598,E2 -9218.598} C_VEL
LIN {X 0,Y 439.351,Z 324.757,A -85,B 0,C 180,E1 -9222.21,E2 -9222.21} C_VEL
LIN {X 0,Y 439.394,Z 324.749,A -85,B 0,C 180,E1 -9225.271,E2 -9225.271} C_VEL
LIN {X 0,Y 439.395,Z 324.752,A -85,B 0,C 180,E1 -9228.743,E2 -9228.743} C_VEL
LIN {X 0,Y 439.378,Z 324.754,A -85,B 0,C 180,E1 -9231.608,E2 -9231.608} C_VEL
LIN {X 0,Y 439.303,Z 324.766,A -85,B 0,C 180,E1 -9233.707,E2 -9233.707} C_VEL
LIN {X 0,Y 439.301,Z 325.326,A -85,B 0,C 180,E1 -9234.836,E2 -9234.836} C_VEL
LIN {X 0,Y 439.241,Z 328.163,A -85,B 0,C 180,E1 -9237.044,E2 -9237.044} C_VEL
LIN {X 0,Y 439.088,Z 332.405,A -85,B 0,C 180,E1 -9240.253,E2 -9240.253} C_VEL
LIN {X 0,Y 438.911,Z 337.107,A -85,B 0,C 180,E1 -9243.727,E2 -9243.727} C_VEL
LIN {X 0,Y 438.799,Z 340.808,A -85,B 0,C 180,E1 -9246.397,E2 -9246.397} C_VEL
LIN {X 0,Y 438.658,Z 345.061,A -85,B 0,C 180,E1 -9249.362,E2 -9249.362} C_VEL
LIN {X 0,Y 438.569,Z 349.388,A -85,B 0,C 180,E1 -9252.274,E2 -9252.274} C_VEL
LIN {X 0,Y 438.539,Z 351.483,A -85,B 0,C 180,E1 -9253.65,E2 -9253.65} C_VEL
LIN {X 0,Y 441.481,Z 364.452,A -85,B 0,C 180,E1 -9254.162,E2 -9254.162} C_VEL
LIN {X 0,Y 442.745,Z 371.85,A -85,B 0,C 180,E1 -9254.522,E2 -9254.522} C_VEL
LIN {X 0,Y 442.274,Z 383.764,A -85,B 0,C 180,E1 -9255.154,E2 -9255.154} C_VEL
LIN {X 0,Y 441.675,Z 395.523,A -85,B 0,C 180,E1 -9255.981,E2 -9255.981} C_VEL
LIN {X 0,Y 441.173,Z 406.079,A -85,B 0,C 180,E1 -9256.924,E2 -9256.924} C_VEL
LIN {X 0,Y 440.519,Z 416.137,A -85,B 0,C 180,E1 -9258.031,E2 -9258.031} C_VEL
LIN {X 0,Y 439.987,Z 424.634,A -85,B 0,C 180,E1 -9259.183,E2 -9259.183} C_VEL
LIN {X 0,Y 439.446,Z 432.888,A -85,B 0,C 180,E1 -9260.566,E2 -9260.566} C_VEL
LIN {X 0,Y 438.981,Z 439.537,A -85,B 0,C 180,E1 -9261.948,E2 -9261.948} C_VEL
LIN {X 0,Y 438.768,Z 443.857,A -85,B 0,C 180,E1 -9263.052,E2 -9263.052} C_VEL
LIN {X 0,Y 438.016,Z 446.287,A -85,B 0,C 180,E1 -9263.748,E2 -9263.748} C_VEL
LIN {X 0,Y 434.993,Z 449.693,A -85,B 0,C 180,E1 -9264.904,E2 -9264.904} C_VEL
LIN {X 0,Y 432.473,Z 451.902,A -85,B 0,C 180,E1 -9265.861,E2 -9265.861} C_VEL
LIN {X 0,Y 431.4,Z 453.27,A -85,B 0,C 180,E1 -9266.614,E2 -9266.614} C_VEL
LIN {X 0,Y 431.317,Z 453.628,A -85,B 0,C 180,E1 -9266.871,E2 -9266.871} C_VEL
LIN {X 0,Y 431.225,Z 455.115,A -85,B 0,C 180,E1 -9268.133,E2 -9268.133} C_VEL
LIN {X 0,Y 431.168,Z 455.964,A -85,B 0,C 180,E1 -9270,E2 -9270} C_VEL
LIN {X 0,Y 431.172,Z 455.777,A -85,B 0,C 180,E1 -9270.934,E2 -9270.934} C_VEL
LIN {X 0,Y 431.327,Z 454.224,A -85,B 0,C 180,E1 -9272.802,E2 -9272.802} C_VEL
LIN {X 0,Y 431.334,Z 452.871,A -85,B 0,C 180,E1 -9273.737,E2 -9273.737} C_VEL
LIN {X 0,Y 431.43,Z 450.009,A -85,B 0,C 180,E1 -9275.141,E2 -9275.141} C_VEL
LIN {X 0,Y 431.656,Z 445.649,A -85,B 0,C 180,E1 -9276.698,E2 -9276.698} C_VEL
LIN {X 0,Y 431.885,Z 441.116,A -85,B 0,C 180,E1 -9277.951,E2 -9277.951} C_VEL
LIN {X 0,Y 432.317,Z 434.808,A -85,B 0,C 180,E1 -9279.356,E2 -9279.356} C_VEL
LIN {X 0,Y 432.846,Z 426.911,A -85,B 0,C 180,E1 -9280.762,E2 -9280.762} C_VEL
LIN {X 0,Y 433.502,Z 417.085,A -85,B 0,C 180,E1 -9282.167,E2 -9282.167} C_VEL
LIN {X 0,Y 434.211,Z 407.453,A -85,B 0,C 180,E1 -9283.266,E2 -9283.266} C_VEL
LIN {X 0,Y 434.719,Z 396.56,A -85,B 0,C 180,E1 -9284.273,E2 -9284.273} C_VEL
LIN {X 0,Y 435.379,Z 385.38,A -85,B 0,C 180,E1 -9285.088,E2 -9285.088} C_VEL
LIN {X 0,Y 435.906,Z 372.799,A -85,B 0,C 180,E1 -9285.788,E2 -9285.788} C_VEL
LIN {X 0,Y 433.564,Z 360.522,A -85,B 0,C 180,E1 -9286.381,E2 -9286.381} C_VEL
LIN {X 0,Y 431.454,Z 351.661,A -85,B 0,C 180,E1 -9286.742,E2 -9286.742} C_VEL
LIN {X 0,Y 431.579,Z 346.833,A -85,B 0,C 180,E1 -9289.997,E2 -9289.997} C_VEL
LIN {X 0,Y 431.662,Z 342.543,A -85,B 0,C 180,E1 -9293.001,E2 -9293.001} C_VEL
LIN {X 0,Y 431.83,Z 338.315,A -85,B 0,C 180,E1 -9296.067,E2 -9296.067} C_VEL
LIN {X 0,Y 431.98,Z 334.107,A -85,B 0,C 180,E1 -9299.214,E2 -9299.214} C_VEL
LIN {X 0,Y 432.172,Z 329.845,A -85,B 0,C 180,E1 -9302.455,E2 -9302.455} C_VEL
LIN {X 0,Y 432.258,Z 326.985,A -85,B 0,C 180,E1 -9304.684,E2 -9304.684} C_VEL
LIN {X 0,Y 432.23,Z 325.647,A -85,B 0,C 180,E1 -9305.828,E2 -9305.828} C_VEL
LIN {X 0,Y 432.337,Z 325.635,A -85,B 0,C 180,E1 -9308.713,E2 -9308.713} C_VEL
LIN {X 0,Y 432.334,Z 325.634,A -85,B 0,C 180,E1 -9311.797,E2 -9311.797} C_VEL
LIN {X 0,Y 432.333,Z 325.629,A -85,B 0,C 180,E1 -9314.347,E2 -9314.347} C_VEL
LIN {X 0,Y 432.3,Z 325.635,A -85,B 0,C 180,E1 -9317.018,E2 -9317.018} C_VEL
LIN {X 0,Y 432.287,Z 325.638,A -85,B 0,C 180,E1 -9319.827,E2 -9319.827} C_VEL
LIN {X 0,Y 432.305,Z 325.637,A -85,B 0,C 180,E1 -9323.022,E2 -9323.022} C_VEL
LIN {X 0,Y 432.358,Z 325.627,A -85,B 0,C 180,E1 -9325.996,E2 -9325.996} C_VEL
LIN {X 0,Y 432.343,Z 325.631,A -85,B 0,C 180,E1 -9329.49,E2 -9329.49} C_VEL
LIN {X 0,Y 432.331,Z 325.63,A -85,B 0,C 180,E1 -9331.873,E2 -9331.873} C_VEL
LIN {X 0,Y 432.372,Z 325.627,A -85,B 0,C 180,E1 -9335.539,E2 -9335.539} C_VEL
LIN {X 0,Y 432.347,Z 325.632,A -85,B 0,C 180,E1 -9339.046,E2 -9339.046} C_VEL
LIN {X 0,Y 432.373,Z 325.624,A -85,B 0,C 180,E1 -9342.011,E2 -9342.011} C_VEL
LIN {X 0,Y 432.388,Z 325.626,A -85,B 0,C 180,E1 -9344.926,E2 -9344.926} C_VEL
LIN {X 0,Y 432.455,Z 325.615,A -85,B 0,C 180,E1 -9347.803,E2 -9347.803} C_VEL
LIN {X 0,Y 432.488,Z 325.611,A -85,B 0,C 180,E1 -9351.59,E2 -9351.59} C_VEL
LIN {X 0,Y 432.594,Z 325.6,A -85,B 0,C 180,E1 -9354.406,E2 -9354.406} C_VEL
LIN {X 0,Y 432.598,Z 325.599,A -85,B 0,C 180,E1 -9358.138,E2 -9358.138} C_VEL
LIN {X 0,Y 432.717,Z 325.585,A -85,B 0,C 180,E1 -9360,E2 -9360} C_VEL
LIN {X 0,Y 432.587,Z 325.601,A -85,B 0,C 180,E1 -9362.794,E2 -9362.794} C_VEL
LIN {X 0,Y 432.569,Z 325.604,A -85,B 0,C 180,E1 -9366.53,E2 -9366.53} C_VEL
LIN {X 0,Y 432.439,Z 325.617,A -85,B 0,C 180,E1 -9369.353,E2 -9369.353} C_VEL
LIN {X 0,Y 432.426,Z 325.617,A -85,B 0,C 180,E1 -9372.803,E2 -9372.803} C_VEL
LIN {X 0,Y 432.408,Z 325.622,A -85,B 0,C 180,E1 -9376.479,E2 -9376.479} C_VEL
LIN {X 0,Y 432.335,Z 325.633,A -85,B 0,C 180,E1 -9379.961,E2 -9379.961} C_VEL
LIN {X 0,Y 432.314,Z 325.633,A -85,B 0,C 180,E1 -9382.965,E2 -9382.965} C_VEL
LIN {X 0,Y 432.334,Z 325.63,A -85,B 0,C 180,E1 -9385.002,E2 -9385.002} C_VEL
LIN {X 0,Y 432.335,Z 325.63,A -85,B 0,C 180,E1 -9388.127,E2 -9388.127} C_VEL
LIN {X 0,Y 432.317,Z 325.636,A -85,B 0,C 180,E1 -9391.346,E2 -9391.346} C_VEL
LIN {X 0,Y 432.338,Z 325.63,A -85,B 0,C 180,E1 -9394.677,E2 -9394.677} C_VEL
LIN {X 0,Y 432.336,Z 325.629,A -85,B 0,C 180,E1 -9398.15,E2 -9398.15} C_VEL
LIN {X 0,Y 432.301,Z 325.634,A -85,B 0,C 180,E1 -9401.801,E2 -9401.801} C_VEL
LIN {X 0,Y 432.331,Z 325.633,A -85,B 0,C 180,E1 -9404.348,E2 -9404.348} C_VEL
LIN {X 0,Y 432.319,Z 325.635,A -85,B 0,C 180,E1 -9407.016,E2 -9407.016} C_VEL
LIN {X 0,Y 432.398,Z 325.81,A -85,B 0,C 180,E1 -9409.668,E2 -9409.668} C_VEL
LIN {X 0,Y 433.278,Z 331.138,A -85,B 0,C 180,E1 -9412.637,E2 -9412.637} C_VEL
LIN {X 0,Y 433.567,Z 335.405,A -85,B 0,C 180,E1 -9414.87,E2 -9414.87} C_VEL
LIN {X 0,Y 433.199,Z 342.102,A -85,B 0,C 180,E1 -9418.18,E2 -9418.18} C_VEL
LIN {X 0,Y 432.845,Z 348.572,A -85,B 0,C 180,E1 -9421.257,E2 -9421.257} C_VEL
LIN {X 0,Y 432.491,Z 355.585,A -85,B 0,C 180,E1 -9424.493,E2 -9424.493} C_VEL
LIN {X 0,Y 432.181,Z 362.307,A -85,B 0,C 180,E1 -9427.534,E2 -9427.534} C_VEL
LIN {X 0,Y 431.932,Z 369.367,A -85,B 0,C 180,E1 -9430.687,E2 -9430.687} C_VEL
LIN {X 0,Y 431.744,Z 375.426,A -85,B 0,C 180,E1 -9433.312,E2 -9433.312} C_VEL
LIN {X 0,Y 434.115,Z 388.768,A -85,B 0,C 180,E1 -9433.789,E2 -9433.789} C_VEL
LIN {X 0,Y 435.612,Z 399.75,A -85,B 0,C 180,E1 -9434.321,E2 -9434.321} C_VEL
LIN {X 0,Y 434.999,Z 411.966,A -85,B 0,C 180,E1 -9435.019,E2 -9435.019} C_VEL
LIN {X 0,Y 434.319,Z 424.421,A -85,B 0,C 180,E1 -9435.952,E2 -9435.952} C_VEL
LIN {X 0,Y 433.621,Z 435.334,A -85,B 0,C 180,E1 -9437.004,E2 -9437.004} C_VEL
LIN {X 0,Y 433.08,Z 444.237,A -85,B 0,C 180,E1 -9438.059,E2 -9438.059} C_VEL
LIN {X 0,Y 432.531,Z 452.42,A -85,B 0,C 180,E1 -9439.23,E2 -9439.23} C_VEL
LIN {X 0,Y 432.066,Z 460.451,A -85,B 0,C 180,E1 -9440.638,E2 -9440.638} C_VEL
LIN {X 0,Y 431.636,Z 466.89,A -85,B 0,C 180,E1 -9442.045,E2 -9442.045} C_VEL
LIN {X 0,Y 431.436,Z 472.32,A -85,B 0,C 180,E1 -9443.555,E2 -9443.555} C_VEL
LIN {X 0,Y 431.288,Z 477.053,A -85,B 0,C 180,E1 -9445.326,E2 -9445.326} C_VEL
LIN {X 0,Y 431.196,Z 478.915,A -85,B 0,C 180,E1 -9446.262,E2 -9446.262} C_VEL
LIN {X 0,Y 431.229,Z 480.314,A -85,B 0,C 180,E1 -9447.197,E2 -9447.197} C_VEL
LIN {X 0,Y 431.199,Z 481.311,A -85,B 0,C 180,E1 -9448.132,E2 -9448.132} C_VEL
LIN {X 0,Y 431.148,Z 481.919,A -85,B 0,C 180,E1 -9449.066,E2 -9449.066} C_VEL
LIN {X 0,Y 431.122,Z 482.135,A -85,B 0,C 180,E1 -9450,E2 -9450} C_VEL
LIN {X 0,Y 431.148,Z 481.92,A -85,B 0,C 180,E1 -9450.934,E2 -9450.934} C_VEL
LIN {X 0,Y 431.199,Z 481.314,A -85,B 0,C 180,E1 -9451.868,E2 -9451.868} C_VEL
LIN {X 0,Y 431.228,Z 480.318,A -85,B 0,C 180,E1 -9452.802,E2 -9452.802} C_VEL
LIN {X 0,Y 431.196,Z 478.92,A -85,B 0,C 180,E1 -9453.738,E2 -9453.738} C_VEL
LIN {X 0,Y 431.33,Z 475.985,A -85,B 0,C 180,E1 -9455.141,E2 -9455.141} C_VEL
LIN {X 0,Y 431.441,Z 472.008,A -85,B 0,C 180,E1 -9456.547,E2 -9456.547} C_VEL
LIN {X 0,Y 431.716,Z 465.896,A -85,B 0,C 180,E1 -9458.189,E2 -9458.189} C_VEL
LIN {X 0,Y 432.137,Z 459.218,A -85,B 0,C 180,E1 -9459.595,E2 -9459.595} C_VEL
LIN {X 0,Y 432.621,Z 450.932,A -85,B 0,C 180,E1 -9461.004,E2 -9461.004} C_VEL
LIN {X 0,Y 433.25,Z 442.445,A -85,B 0,C 180,E1 -9462.173,E2 -9462.173} C_VEL
LIN {X 0,Y 433.87,Z 432.324,A -85,B 0,C 180,E1 -9463.308,E2 -9463.308} C_VEL
LIN {X 0,Y 434.481,Z 421.58,A -85,B 0,C 180,E1 -9464.28,E2 -9464.28} C_VEL
LIN {X 0,Y 435.112,Z 410.208,A -85,B 0,C 180,E1 -9465.096,E2 -9465.096} C_VEL
LIN {X 0,Y 435.563,Z 398.546,A -85,B 0,C 180,E1 -9465.74,E2 -9465.74} C_VEL
LIN {X 0,Y 433.63,Z 385.575,A -85,B 0,C 180,E1 -9466.337,E2 -9466.337} C_VEL
LIN {X 0,Y 431.736,Z 375.25,A -85,B 0,C 180,E1 -9466.71,E2 -9466.71} C_VEL
LIN {X 0,Y 431.979,Z 367.874,A -85,B 0,C 180,E1 -9469.977,E2 -9469.977} C_VEL
LIN {X 0,Y 432.296,Z 360.082,A -85,B 0,C 180,E1 -9473.471,E2 -9473.471} C_VEL
LIN {X 0,Y 432.618,Z 353.001,A -85,B 0,C 180,E1 -9476.685,E2 -9476.685} C_VEL
LIN {X 0,Y 432.96,Z 346.578,A -85,B 0,C 180,E1 -9479.675,E2 -9479.675} C_VEL
LIN {X 0,Y 433.229,Z 340.738,A -85,B 0,C 180,E1 -9482.481,E2 -9482.481} C_VEL
LIN {X 0,Y 433.567,Z 335.4,A -85,B 0,C 180,E1 -9485.13,E2 -9485.13} C_VEL
LIN {X 0,Y 433.276,Z 331.126,A -85,B 0,C 180,E1 -9487.363,E2 -9487.363} C_VEL
LIN {X 0,Y 432.42,Z 325.626,A -85,B 0,C 180,E1 -9490.441,E2 -9490.441} C_VEL
LIN {X 0,Y 432.373,Z 325.629,A -85,B 0,C 180,E1 -9494.341,E2 -9494.341} C_VEL
LIN {X 0,Y 432.302,Z 325.634,A -85,B 0,C 180,E1 -9498.199,E2 -9498.199} C_VEL
LIN {X 0,Y 432.323,Z 325.632,A -85,B 0,C 180,E1 -9501.286,E2 -9501.286} C_VEL
LIN {X 0,Y 432.338,Z 325.634,A -85,B 0,C 180,E1 -9504.367,E2 -9504.367} C_VEL
LIN {X 0,Y 432.315,Z 325.633,A -85,B 0,C 180,E1 -9507.556,E2 -9507.556} C_VEL
LIN {X 0,Y 432.318,Z 325.635,A -85,B 0,C 180,E1 -9510.811,E2 -9510.811} C_VEL
LIN {X 0,Y 432.316,Z 325.633,A -85,B 0,C 180,E1 -9513.964,E2 -9513.964} C_VEL
LIN {X 0,Y 432.358,Z 325.63,A -85,B 0,C 180,E1 -9516.023,E2 -9516.023} C_VEL
LIN {X 0,Y 432.341,Z 325.63,A -85,B 0,C 180,E1 -9519.046,E2 -9519.046} C_VEL
LIN {X 0,Y 432.368,Z 325.629,A -85,B 0,C 180,E1 -9522.011,E2 -9522.011} C_VEL
LIN {X 0,Y 432.382,Z 325.624,A -85,B 0,C 180,E1 -9524.926,E2 -9524.926} C_VEL
LIN {X 0,Y 432.449,Z 325.618,A -85,B 0,C 180,E1 -9527.803,E2 -9527.803} C_VEL
LIN {X 0,Y 432.482,Z 325.615,A -85,B 0,C 180,E1 -9531.59,E2 -9531.59} C_VEL
LIN {X 0,Y 432.594,Z 325.6,A -85,B 0,C 180,E1 -9534.406,E2 -9534.406} C_VEL
LIN {X 0,Y 432.594,Z 325.6,A -85,B 0,C 180,E1 -9538.138,E2 -9538.138} C_VEL
LIN {X 0,Y 432.714,Z 325.585,A -85,B 0,C 180,E1 -9540,E2 -9540} C_VEL
LIN {X 0,Y 432.583,Z 325.598,A -85,B 0,C 180,E1 -9542.794,E2 -9542.794} C_VEL
LIN {X 0,Y 432.565,Z 325.601,A -85,B 0,C 180,E1 -9546.531,E2 -9546.531} C_VEL
LIN {X 0,Y 432.433,Z 325.621,A -85,B 0,C 180,E1 -9549.353,E2 -9549.353} C_VEL
LIN {X 0,Y 432.42,Z 325.621,A -85,B 0,C 180,E1 -9552.804,E2 -9552.804} C_VEL
LIN {X 0,Y 432.403,Z 325.62,A -85,B 0,C 180,E1 -9556.479,E2 -9556.479} C_VEL
LIN {X 0,Y 432.33,Z 325.631,A -85,B 0,C 180,E1 -9559.961,E2 -9559.961} C_VEL
LIN {X 0,Y 432.308,Z 325.636,A -85,B 0,C 180,E1 -9562.965,E2 -9562.965} C_VEL
LIN {X 0,Y 432.33,Z 325.633,A -85,B 0,C 180,E1 -9565.003,E2 -9565.003} C_VEL
LIN {X 0,Y 432.33,Z 325.63,A -85,B 0,C 180,E1 -9568.127,E2 -9568.127} C_VEL
LIN {X 0,Y 432.312,Z 325.633,A -85,B 0,C 180,E1 -9571.347,E2 -9571.347} C_VEL
LIN {X 0,Y 432.334,Z 325.634,A -85,B 0,C 180,E1 -9574.678,E2 -9574.678} C_VEL
LIN {X 0,Y 432.324,Z 325.633,A -85,B 0,C 180,E1 -9578.152,E2 -9578.152} C_VEL
LIN {X 0,Y 432.302,Z 325.634,A -85,B 0,C 180,E1 -9581.801,E2 -9581.801} C_VEL
LIN {X 0,Y 432.328,Z 325.634,A -85,B 0,C 180,E1 -9584.348,E2 -9584.348} C_VEL
LIN {X 0,Y 432.316,Z 325.633,A -85,B 0,C 180,E1 -9587.017,E2 -9587.017} C_VEL
LIN {X 0,Y 432.352,Z 325.629,A -85,B 0,C 180,E1 -9589.818,E2 -9589.818} C_VEL
LIN {X 0,Y 432.29,Z 325.641,A -85,B 0,C 180,E1 -9593.022,E2 -9593.022} C_VEL
LIN {X 0,Y 432.209,Z 325.723,A -85,B 0,C 180,E1 -9594.394,E2 -9594.394} C_VEL
LIN {X 0,Y 432.228,Z 328.287,A -85,B 0,C 180,E1 -9596.439,E2 -9596.439} C_VEL
LIN {X 0,Y 432.082,Z 332.542,A -85,B 0,C 180,E1 -9599.721,E2 -9599.721} C_VEL
LIN {X 0,Y 431.855,Z 336.768,A -85,B 0,C 180,E1 -9602.893,E2 -9602.893} C_VEL
LIN {X 0,Y 431.785,Z 340.979,A -85,B 0,C 180,E1 -9605.99,E2 -9605.99} C_VEL
LIN {X 0,Y 431.592,Z 345.248,A -85,B 0,C 180,E1 -9609.008,E2 -9609.008} C_VEL
LIN {X 0,Y 431.503,Z 349.588,A -85,B 0,C 180,E1 -9611.974,E2 -9611.974} C_VEL
LIN {X 0,Y 431.499,Z 351.814,A -85,B 0,C 180,E1 -9613.38,E2 -9613.38} C_VEL
LIN {X 0,Y 434.501,Z 365.025,A -85,B 0,C 180,E1 -9613.914,E2 -9613.914} C_VEL
LIN {X 0,Y 435.892,Z 373.369,A -85,B 0,C 180,E1 -9614.333,E2 -9614.333} C_VEL
LIN {X 0,Y 435.344,Z 385.773,A -85,B 0,C 180,E1 -9615.032,E2 -9615.032} C_VEL
LIN {X 0,Y 434.731,Z 396.878,A -85,B 0,C 180,E1 -9615.847,E2 -9615.847} C_VEL
LIN {X 0,Y 434.142,Z 408.189,A -85,B 0,C 180,E1 -9616.902,E2 -9616.902} C_VEL
LIN {X 0,Y 433.413,Z 418.168,A -85,B 0,C 180,E1 -9618.069,E2 -9618.069} C_VEL
LIN {X 0,Y 432.766,Z 427.811,A -85,B 0,C 180,E1 -9619.474,E2 -9619.474} C_VEL
LIN {X 0,Y 432.26,Z 435.503,A -85,B 0,C 180,E1 -9620.879,E2 -9620.879} C_VEL
LIN {X 0,Y 431.784,Z 442.561,A -85,B 0,C 180,E1 -9622.519,E2 -9622.519} C_VEL
LIN {X 0,Y 431.632,Z 447.258,A -85,B 0,C 180,E1 -9623.925,E2 -9623.925} C_VEL
LIN {X 0,Y 431.36,Z 450.86,A -85,B 0,C 180,E1 -9625.328,E2 -9625.328} C_VEL
LIN {X 0,Y 431.317,Z 453.628,A -85,B 0,C 180,E1 -9626.871,E2 -9626.871} C_VEL
LIN {X 0,Y 430.64,Z 454.684,A -85,B 0,C 180,E1 -9627.639,E2 -9627.639} C_VEL
LIN {X 0,Y 427.71,Z 455.898,A -85,B 0,C 180,E1 -9628.894,E2 -9628.894} C_VEL
LIN {X 0,Y 425.234,Z 456.265,A -85,B 0,C 180,E1 -9629.913,E2 -9629.913} C_VEL
LIN {X 0,Y 424.174,Z 456.12,A -85,B 0,C 180,E1 -9630.702,E2 -9630.702} C_VEL
LIN {X 0,Y 424.092,Z 455.98,A -85,B 0,C 180,E1 -9630.969,E2 -9630.969} C_VEL
LIN {X 0,Y 424.241,Z 454.439,A -85,B 0,C 180,E1 -9632.849,E2 -9632.849} C_VEL
LIN {X 0,Y 424.241,Z 453.086,A -85,B 0,C 180,E1 -9633.8,E2 -9633.8} C_VEL
LIN {X 0,Y 424.379,Z 450.223,A -85,B 0,C 180,E1 -9635.226,E2 -9635.226} C_VEL
LIN {X 0,Y 424.584,Z 446.197,A -85,B 0,C 180,E1 -9636.702,E2 -9636.702} C_VEL
LIN {X 0,Y 424.854,Z 441.33,A -85,B 0,C 180,E1 -9638.083,E2 -9638.083} C_VEL
LIN {X 0,Y 425.317,Z 435.021,A -85,B 0,C 180,E1 -9639.511,E2 -9639.511} C_VEL
LIN {X 0,Y 425.877,Z 427.123,A -85,B 0,C 180,E1 -9640.94,E2 -9640.94} C_VEL
LIN {X 0,Y 426.423,Z 419.072,A -85,B 0,C 180,E1 -9642.131,E2 -9642.131} C_VEL
LIN {X 0,Y 427.202,Z 409.24,A -85,B 0,C 180,E1 -9643.316,E2 -9643.316} C_VEL
LIN {X 0,Y 427.699,Z 399.573,A -85,B 0,C 180,E1 -9644.27,E2 -9644.27} C_VEL
LIN {X 0,Y 428.311,Z 389.108,A -85,B 0,C 180,E1 -9645.099,E2 -9645.099} C_VEL
LIN {X 0,Y 428.977,Z 376.5,A -85,B 0,C 180,E1 -9645.866,E2 -9645.866} C_VEL
LIN {X 0,Y 428.771,Z 371.717,A -85,B 0,C 180,E1 -9646.119,E2 -9646.119} C_VEL
LIN {X 0,Y 426.238,Z 359.53,A -85,B 0,C 180,E1 -9646.711,E2 -9646.711} C_VEL
LIN {X 0,Y 424.367,Z 351.877,A -85,B 0,C 180,E1 -9647.024,E2 -9647.024} C_VEL
LIN {X 0,Y 424.505,Z 348.456,A -85,B 0,C 180,E1 -9649.337,E2 -9649.337} C_VEL
LIN {X 0,Y 424.58,Z 344.161,A -85,B 0,C 180,E1 -9652.378,E2 -9652.378} C_VEL
LIN {X 0,Y 424.728,Z 339.887,A -85,B 0,C 180,E1 -9655.482,E2 -9655.482} C_VEL
LIN {X 0,Y 424.903,Z 335.534,A -85,B 0,C 180,E1 -9658.761,E2 -9658.761} C_VEL
LIN {X 0,Y 425.091,Z 331.407,A -85,B 0,C 180,E1 -9661.941,E2 -9661.941} C_VEL
LIN {X 0,Y 425.22,Z 328.444,A -85,B 0,C 180,E1 -9664.269,E2 -9664.269} C_VEL
LIN {X 0,Y 425.185,Z 326.525,A -85,B 0,C 180,E1 -9665.91,E2 -9665.91} C_VEL
LIN {X 0,Y 425.278,Z 326.512,A -85,B 0,C 180,E1 -9669.04,E2 -9669.04} C_VEL
LIN {X 0,Y 425.29,Z 326.511,A -85,B 0,C 180,E1 -9671.958,E2 -9671.958} C_VEL
LIN {X 0,Y 425.283,Z 326.51,A -85,B 0,C 180,E1 -9675.283,E2 -9675.283} C_VEL
LIN {X 0,Y 425.245,Z 326.513,A -85,B 0,C 180,E1 -9678.618,E2 -9678.618} C_VEL
LIN {X 0,Y 425.279,Z 326.512,A -85,B 0,C 180,E1 -9681.099,E2 -9681.099} C_VEL
LIN {X 0,Y 425.298,Z 326.507,A -85,B 0,C 180,E1 -9684.664,E2 -9684.664} C_VEL
LIN {X 0,Y 425.262,Z 326.51,A -85,B 0,C 180,E1 -9688.073,E2 -9688.073} C_VEL
LIN {X 0,Y 425.301,Z 326.508,A -85,B 0,C 180,E1 -9691.366,E2 -9691.366} C_VEL
LIN {X 0,Y 425.263,Z 326.513,A -85,B 0,C 180,E1 -9694.552,E2 -9694.552} C_VEL
LIN {X 0,Y 425.299,Z 326.51,A -85,B 0,C 180,E1 -9696.634,E2 -9696.634} C_VEL
LIN {X 0,Y 425.325,Z 326.504,A -85,B 0,C 180,E1 -9700.364,E2 -9700.364} C_VEL
LIN {X 0,Y 425.384,Z 326.494,A -85,B 0,C 180,E1 -9703.688,E2 -9703.688} C_VEL
LIN {X 0,Y 425.408,Z 326.493,A -85,B 0,C 180,E1 -9707.598,E2 -9707.598} C_VEL
LIN {X 0,Y 425.438,Z 326.489,A -85,B 0,C 180,E1 -9711.45,E2 -9711.45} C_VEL
LIN {X 0,Y 425.551,Z 326.477,A -85,B 0,C 180,E1 -9714.313,E2 -9714.313} C_VEL
LIN {X 0,Y 425.567,Z 326.475,A -85,B 0,C 180,E1 -9718.107,E2 -9718.107} C_VEL
LIN {X 0,Y 425.687,Z 326.46,A -85,B 0,C 180,E1 -9720,E2 -9720} C_VEL
LIN {X 0,Y 425.54,Z 326.478,A -85,B 0,C 180,E1 -9722.84,E2 -9722.84} C_VEL
LIN {X 0,Y 425.526,Z 326.48,A -85,B 0,C 180,E1 -9726.639,E2 -9726.639} C_VEL
LIN {X 0,Y 425.397,Z 326.495,A -85,B 0,C 180,E1 -9729.509,E2 -9729.509} C_VEL
LIN {X 0,Y 425.389,Z 326.494,A -85,B 0,C 180,E1 -9732.903,E2 -9732.903} C_VEL
LIN {X 0,Y 425.357,Z 326.5,A -85,B 0,C 180,E1 -9736.605,E2 -9736.605} C_VEL
LIN {X 0,Y 425.325,Z 326.506,A -85,B 0,C 180,E1 -9739.636,E2 -9739.636} C_VEL
LIN {X 0,Y 425.301,Z 326.508,A -85,B 0,C 180,E1 -9743.365,E2 -9743.365} C_VEL
LIN {X 0,Y 425.292,Z 326.505,A -85,B 0,C 180,E1 -9746.499,E2 -9746.499} C_VEL
LIN {X 0,Y 425.28,Z 326.511,A -85,B 0,C 180,E1 -9749.72,E2 -9749.72} C_VEL
LIN {X 0,Y 425.28,Z 326.512,A -85,B 0,C 180,E1 -9753.048,E2 -9753.048} C_VEL
LIN {X 0,Y 425.282,Z 326.51,A -85,B 0,C 180,E1 -9755.929,E2 -9755.929} C_VEL
LIN {X 0,Y 425.263,Z 326.513,A -85,B 0,C 180,E1 -9759.038,E2 -9759.038} C_VEL
LIN {X 0,Y 425.254,Z 326.513,A -85,B 0,C 180,E1 -9762.656,E2 -9762.656} C_VEL
LIN {X 0,Y 425.283,Z 326.511,A -85,B 0,C 180,E1 -9765.283,E2 -9765.283} C_VEL
LIN {X 0,Y 425.279,Z 326.512,A -85,B 0,C 180,E1 -9768.622,E2 -9768.622} C_VEL
LIN {X 0,Y 425.31,Z 326.546,A -85,B 0,C 180,E1 -9769.321,E2 -9769.321} C_VEL
LIN {X 0,Y 426.246,Z 331.951,A -85,B 0,C 180,E1 -9772.406,E2 -9772.406} C_VEL
LIN {X 0,Y 426.578,Z 336.405,A -85,B 0,C 180,E1 -9774.786,E2 -9774.786} C_VEL
LIN {X 0,Y 426.191,Z 343.095,A -85,B 0,C 180,E1 -9778.151,E2 -9778.151} C_VEL
LIN {X 0,Y 425.792,Z 349.819,A -85,B 0,C 180,E1 -9781.402,E2 -9781.402} C_VEL
LIN {X 0,Y 425.419,Z 356.56,A -85,B 0,C 180,E1 -9784.563,E2 -9784.563} C_VEL
LIN {X 0,Y 425.096,Z 363.567,A -85,B 0,C 180,E1 -9787.795,E2 -9787.795} C_VEL
LIN {X 0,Y 424.814,Z 371.014,A -85,B 0,C 180,E1 -9791.18,E2 -9791.18} C_VEL
LIN {X 0,Y 424.675,Z 375.032,A -85,B 0,C 180,E1 -9793,E2 -9793} C_VEL
LIN {X 0,Y 427.429,Z 390.864,A -85,B 0,C 180,E1 -9793.621,E2 -9793.621} C_VEL
LIN {X 0,Y 428.735,Z 400.666,A -85,B 0,C 180,E1 -9794.124,E2 -9794.124} C_VEL
LIN {X 0,Y 428.035,Z 413.519,A -85,B 0,C 180,E1 -9794.891,E2 -9794.891} C_VEL
LIN {X 0,Y 427.337,Z 425.234,A -85,B 0,C 180,E1 -9795.813,E2 -9795.813} C_VEL
LIN {X 0,Y 426.597,Z 436.19,A -85,B 0,C 180,E1 -9796.907,E2 -9796.907} C_VEL
LIN {X 0,Y 426.001,Z 445.81,A -85,B 0,C 180,E1 -9798.099,E2 -9798.099} C_VEL
LIN {X 0,Y 425.45,Z 453.695,A -85,B 0,C 180,E1 -9799.29,E2 -9799.29} C_VEL
LIN {X 0,Y 424.945,Z 461.397,A -85,B 0,C 180,E1 -9800.72,E2 -9800.72} C_VEL
LIN {X 0,Y 424.487,Z 468.497,A -85,B 0,C 180,E1 -9802.388,E2 -9802.388} C_VEL
LIN {X 0,Y 424.271,Z 473.618,A -85,B 0,C 180,E1 -9803.951,E2 -9803.951} C_VEL
LIN {X 0,Y 424.219,Z 476.838,A -85,B 0,C 180,E1 -9805.248,E2 -9805.248} C_VEL
LIN {X 0,Y 424.107,Z 478.699,A -85,B 0,C 180,E1 -9806.199,E2 -9806.199} C_VEL
LIN {X 0,Y 424.126,Z 480.098,A -85,B 0,C 180,E1 -9807.15,E2 -9807.15} C_VEL
LIN {X 0,Y 424.125,Z 481.096,A -85,B 0,C 180,E1 -9808.1,E2 -9808.1} C_VEL
LIN {X 0,Y 424.069,Z 481.704,A -85,B 0,C 180,E1 -9809.05,E2 -9809.05} C_VEL
LIN {X 0,Y 424.041,Z 481.92,A -85,B 0,C 180,E1 -9810,E2 -9810} C_VEL
LIN {X 0,Y 424.125,Z 481.099,A -85,B 0,C 180,E1 -9811.899,E2 -9811.899} C_VEL
LIN {X 0,Y 424.125,Z 480.103,A -85,B 0,C 180,E1 -9812.849,E2 -9812.849} C_VEL
LIN {X 0,Y 424.107,Z 478.704,A -85,B 0,C 180,E1 -9813.8,E2 -9813.8} C_VEL
LIN {X 0,Y 424.246,Z 475.769,A -85,B 0,C 180,E1 -9815.227,E2 -9815.227} C_VEL
LIN {X 0,Y 424.359,Z 471.792,A -85,B 0,C 180,E1 -9816.657,E2 -9816.657} C_VEL
LIN {X 0,Y 424.666,Z 465.68,A -85,B 0,C 180,E1 -9818.326,E2 -9818.326} C_VEL
LIN {X 0,Y 425.086,Z 459.001,A -85,B 0,C 180,E1 -9819.756,E2 -9819.756} C_VEL
LIN {X 0,Y 425.628,Z 450.716,A -85,B 0,C 180,E1 -9821.187,E2 -9821.187} C_VEL
LIN {X 0,Y 426.3,Z 442.23,A -85,B 0,C 180,E1 -9822.375,E2 -9822.375} C_VEL
LIN {X 0,Y 426.916,Z 432.533,A -85,B 0,C 180,E1 -9823.485,E2 -9823.485} C_VEL
LIN {X 0,Y 427.568,Z 421.363,A -85,B 0,C 180,E1 -9824.516,E2 -9824.516} C_VEL
LIN {X 0,Y 428.252,Z 409.992,A -85,B 0,C 180,E1 -9825.344,E2 -9825.344} C_VEL
LIN {X 0,Y 428.684,Z 399.538,A -85,B 0,C 180,E1 -9825.938,E2 -9825.938} C_VEL
LIN {X 0,Y 426.738,Z 386.483,A -85,B 0,C 180,E1 -9826.571,E2 -9826.571} C_VEL
LIN {X 0,Y 424.673,Z 375.033,A -85,B 0,C 180,E1 -9826.999,E2 -9826.999} C_VEL
LIN {X 0,Y 424.935,Z 367.707,A -85,B 0,C 180,E1 -9830.323,E2 -9830.323} C_VEL
LIN {X 0,Y 425.267,Z 359.923,A -85,B 0,C 180,E1 -9833.883,E2 -9833.883} C_VEL
LIN {X 0,Y 425.666,Z 352.049,A -85,B 0,C 180,E1 -9837.534,E2 -9837.534} C_VEL
LIN {X 0,Y 426.064,Z 344.948,A -85,B 0,C 180,E1 -9840.935,E2 -9840.935} C_VEL
LIN {X 0,Y 426.514,Z 337.742,A -85,B 0,C 180,E1 -9844.524,E2 -9844.524} C_VEL
LIN {X 0,Y 426.367,Z 333.065,A -85,B 0,C 180,E1 -9846.986,E2 -9846.986} C_VEL
LIN {X 0,Y 425.546,Z 327.51,A -85,B 0,C 180,E1 -9850.096,E2 -9850.096} C_VEL
LIN {X 0,Y 425.35,Z 326.508,A -85,B 0,C 180,E1 -9850.741,E2 -9850.741} C_VEL
LIN {X 0,Y 425.33,Z 326.51,A -85,B 0,C 180,E1 -9853.945,E2 -9853.945} C_VEL
LIN {X 0,Y 425.254,Z 326.513,A -85,B 0,C 180,E1 -9857.344,E2 -9857.344} C_VEL
LIN {X 0,Y 425.258,Z 326.514,A -85,B 0,C 180,E1 -9860.961,E2 -9860.961} C_VEL
LIN {X 0,Y 425.277,Z 326.51,A -85,B 0,C 180,E1 -9864.07,E2 -9864.07} C_VEL
LIN {X 0,Y 425.274,Z 326.513,A -85,B 0,C 180,E1 -9866.951,E2 -9866.951} C_VEL
LIN {X 0,Y 425.274,Z 326.512,A -85,B 0,C 180,E1 -9870.279,E2 -9870.279} C_VEL
LIN {X 0,Y 425.288,Z 326.506,A -85,B 0,C 180,E1 -9873.501,E2 -9873.501} C_VEL
LIN {X 0,Y 425.296,Z 326.509,A -85,B 0,C 180,E1 -9876.634,E2 -9876.634} C_VEL
LIN {X 0,Y 425.319,Z 326.507,A -85,B 0,C 180,E1 -9880.364,E2 -9880.364} C_VEL
LIN {X 0,Y 425.378,Z 326.499,A -85,B 0,C 180,E1 -9883.688,E2 -9883.688} C_VEL
LIN {X 0,Y 425.402,Z 326.494,A -85,B 0,C 180,E1 -9887.598,E2 -9887.598} C_VEL
LIN {X 0,Y 425.432,Z 326.491,A -85,B 0,C 180,E1 -9891.45,E2 -9891.45} C_VEL
LIN {X 0,Y 425.569,Z 326.475,A -85,B 0,C 180,E1 -9894.313,E2 -9894.313} C_VEL
LIN {X 0,Y 425.563,Z 326.476,A -85,B 0,C 180,E1 -9898.107,E2 -9898.107} C_VEL
LIN {X 0,Y 425.683,Z 326.461,A -85,B 0,C 180,E1 -9900,E2 -9900} C_VEL
LIN {X 0,Y 425.537,Z 326.475,A -85,B 0,C 180,E1 -9902.84,E2 -9902.84} C_VEL
LIN {X 0,Y 425.523,Z 326.478,A -85,B 0,C 180,E1 -9906.639,E2 -9906.639} C_VEL
LIN {X 0,Y 425.391,Z 326.498,A -85,B 0,C 180,E1 -9909.51,E2 -9909.51} C_VEL
LIN {X 0,Y 425.383,Z 326.498,A -85,B 0,C 180,E1 -9912.904,E2 -9912.904} C_VEL
LIN {X 0,Y 425.352,Z 326.499,A -85,B 0,C 180,E1 -9916.605,E2 -9916.605} C_VEL
LIN {X 0,Y 425.319,Z 326.505,A -85,B 0,C 180,E1 -9919.636,E2 -9919.636} C_VEL
LIN {X 0,Y 425.296,Z 326.51,A -85,B 0,C 180,E1 -9923.366,E2 -9923.366} C_VEL
LIN {X 0,Y 425.288,Z 326.51,A -85,B 0,C 180,E1 -9926.499,E2 -9926.499} C_VEL
LIN {X 0,Y 425.274,Z 326.508,A -85,B 0,C 180,E1 -9929.721,E2 -9929.721} C_VEL
LIN {X 0,Y 425.275,Z 326.512,A -85,B 0,C 180,E1 -9933.049,E2 -9933.049} C_VEL
LIN {X 0,Y 425.276,Z 326.509,A -85,B 0,C 180,E1 -9935.93,E2 -9935.93} C_VEL
LIN {X 0,Y 425.256,Z 326.515,A -85,B 0,C 180,E1 -9939.038,E2 -9939.038} C_VEL
LIN {X 0,Y 425.254,Z 326.517,A -85,B 0,C 180,E1 -9942.656,E2 -9942.656} C_VEL
LIN {X 0,Y 425.28,Z 326.507,A -85,B 0,C 180,E1 -9945.284,E2 -9945.284} C_VEL
LIN {X 0,Y 425.3,Z 326.509,A -85,B 0,C 180,E1 -9948.626,E2 -9948.626} C_VEL
LIN {X 0,Y 425.316,Z 326.505,A -85,B 0,C 180,E1 -9951.105,E2 -9951.105} C_VEL
LIN {X 0,Y 425.167,Z 326.526,A -85,B 0,C 180,E1 -9954.093,E2 -9954.093} C_VEL
LIN {X 0,Y 425.23,Z 328.412,A -85,B 0,C 180,E1 -9955.811,E2 -9955.811} C_VEL
LIN {X 0,Y 425.019,Z 332.854,A -85,B 0,C 180,E1 -9959.301,E2 -9959.301} C_VEL
LIN {X 0,Y 424.835,Z 336.923,A -85,B 0,C 180,E1 -9962.407,E2 -9962.407} C_VEL
LIN {X 0,Y 424.715,Z 341.152,A -85,B 0,C 180,E1 -9965.564,E2 -9965.564} C_VEL
LIN {X 0,Y 424.561,Z 345.435,A -85,B 0,C 180,E1 -9968.644,E2 -9968.644} C_VEL
LIN {X 0,Y 424.455,Z 349.789,A -85,B 0,C 180,E1 -9971.664,E2 -9971.664} C_VEL
LIN {X 0,Y 424.429,Z 351.886,A -85,B 0,C 180,E1 -9973.081,E2 -9973.081} C_VEL
LIN {X 0,Y 427.765,Z 366.604,A -85,B 0,C 180,E1 -9973.708,E2 -9973.708} C_VEL
LIN {X 0,Y 429.047,Z 373.595,A -85,B 0,C 180,E1 -9974.076,E2 -9974.076} C_VEL
LIN {X 0,Y 428.494,Z 385.995,A -85,B 0,C 180,E1 -9974.787,E2 -9974.787} C_VEL
LIN {X 0,Y 427.865,Z 397.098,A -85,B 0,C 180,E1 -9975.616,E2 -9975.616} C_VEL
LIN {X 0,Y 427.24,Z 408.408,A -85,B 0,C 180,E1 -9976.686,E2 -9976.686} C_VEL
LIN {X 0,Y 426.47,Z 418.387,A -85,B 0,C 180,E1 -9977.872,E2 -9977.872} C_VEL
LIN {X 0,Y 425.788,Z 428.029,A -85,B 0,C 180,E1 -9979.299,E2 -9979.299} C_VEL
LIN {X 0,Y 425.255,Z 435.721,A -85,B 0,C 180,E1 -9980.728,E2 -9980.728} C_VEL
LIN {X 0,Y 424.741,Z 442.778,A -85,B 0,C 180,E1 -9982.394,E2 -9982.394} C_VEL
LIN {X 0,Y 424.577,Z 446.861,A -85,B 0,C 180,E1 -9983.616,E2 -9983.616} C_VEL
LIN {X 0,Y 424.293,Z 451.076,A -85,B 0,C 180,E1 -9985.25,E2 -9985.25} C_VEL
LIN {X 0,Y 424.23,Z 453.914,A -85,B 0,C 180,E1 -9986.867,E2 -9986.867} C_VEL
LIN {X 0,Y 424.152,Z 455.331,A -85,B 0,C 180,E1 -9988.101,E2 -9988.101} C_VEL
LIN {X 0,Y 424.085,Z 456.179,A -85,B 0,C 180,E1 -9990,E2 -9990} C_VEL
LIN {X 0,Y 424.092,Z 455.98,A -85,B 0,C 180,E1 -9990.969,E2 -9990.969} C_VEL
LIN {X 0,Y 423.428,Z 455.548,A -85,B 0,C 180,E1 -9991.759,E2 -9991.759} C_VEL
LIN {X 0,Y 420.58,Z 454.357,A -85,B 0,C 180,E1 -9993.04,E2 -9993.04} C_VEL
LIN {X 0,Y 418.231,Z 452.908,A -85,B 0,C 180,E1 -9994.063,E2 -9994.063} C_VEL
LIN {X 0,Y 417.309,Z 451.464,A -85,B 0,C 180,E1 -9994.843,E2 -9994.843} C_VEL
LIN {X 0,Y 417.28,Z 450.898,A -85,B 0,C 180,E1 -9995.104,E2 -9995.104} C_VEL
LIN {X 0,Y 417.521,Z 446.554,A -85,B 0,C 180,E1 -9996.767,E2 -9996.767} C_VEL
LIN {X 0,Y 417.818,Z 441.544,A -85,B 0,C 180,E1 -9998.22,E2 -9998.22} C_VEL
LIN {X 0,Y 418.323,Z 435.234,A -85,B 0,C 180,E1 -9999.672,E2 -9999.672} C_VEL
LIN {X 0,Y 418.912,Z 427.335,A -85,B 0,C 180,E1 -10001.124,E2 -10001.124} C_VEL
LIN {X 0,Y 419.48,Z 419.284,A -85,B 0,C 180,E1 -10002.334,E2 -10002.334} C_VEL
LIN {X 0,Y 420.299,Z 409.451,A -85,B 0,C 180,E1 -10003.539,E2 -10003.539} C_VEL
LIN {X 0,Y 420.92,Z 398.4,A -85,B 0,C 180,E1 -10004.628,E2 -10004.628} C_VEL
LIN {X 0,Y 421.559,Z 387.558,A -85,B 0,C 180,E1 -10005.471,E2 -10005.471} C_VEL
LIN {X 0,Y 422.213,Z 374.655,A -85,B 0,C 180,E1 -10006.241,E2 -10006.241} C_VEL
LIN {X 0,Y 419.808,Z 362.624,A -85,B 0,C 180,E1 -10006.875,E2 -10006.875} C_VEL
LIN {X 0,Y 417.324,Z 352.08,A -85,B 0,C 180,E1 -10007.323,E2 -10007.323} C_VEL
LIN {X 0,Y 417.446,Z 348.653,A -85,B 0,C 180,E1 -10009.677,E2 -10009.677} C_VEL
LIN {X 0,Y 417.519,Z 344.345,A -85,B 0,C 180,E1 -10012.777,E2 -10012.777} C_VEL
LIN {X 0,Y 417.703,Z 340.054,A -85,B 0,C 180,E1 -10015.942,E2 -10015.942} C_VEL
LIN {X 0,Y 417.873,Z 335.82,A -85,B 0,C 180,E1 -10019.192,E2 -10019.192} C_VEL
LIN {X 0,Y 418.102,Z 331.536,A -85,B 0,C 180,E1 -10022.54,E2 -10022.54} C_VEL
LIN {X 0,Y 418.164,Z 328.665,A -85,B 0,C 180,E1 -10024.85,E2 -10024.85} C_VEL
LIN {X 0,Y 418.177,Z 327.399,A -85,B 0,C 180,E1 -10026.225,E2 -10026.225} C_VEL
LIN {X 0,Y 418.244,Z 327.388,A -85,B 0,C 180,E1 -10029.379,E2 -10029.379} C_VEL
LIN {X 0,Y 418.229,Z 327.387,A -85,B 0,C 180,E1 -10032.321,E2 -10032.321} C_VEL
LIN {X 0,Y 418.234,Z 327.387,A -85,B 0,C 180,E1 -10035.108,E2 -10035.108} C_VEL
LIN {X 0,Y 418.217,Z 327.391,A -85,B 0,C 180,E1 -10037.764,E2 -10037.764} C_VEL
LIN {X 0,Y 418.236,Z 327.389,A -85,B 0,C 180,E1 -10041.556,E2 -10041.556} C_VEL
LIN {X 0,Y 418.258,Z 327.386,A -85,B 0,C 180,E1 -10045.159,E2 -10045.159} C_VEL
LIN {X 0,Y 418.243,Z 327.388,A -85,B 0,C 180,E1 -10047.471,E2 -10047.471} C_VEL
LIN {X 0,Y 418.258,Z 327.386,A -85,B 0,C 180,E1 -10050.897,E2 -10050.897} C_VEL
LIN {X 0,Y 418.229,Z 327.387,A -85,B 0,C 180,E1 -10054.093,E2 -10054.093} C_VEL
LIN {X 0,Y 418.234,Z 327.39,A -85,B 0,C 180,E1 -10057.263,E2 -10057.263} C_VEL
LIN {X 0,Y 418.28,Z 327.382,A -85,B 0,C 180,E1 -10060.364,E2 -10060.364} C_VEL
LIN {X 0,Y 418.313,Z 327.376,A -85,B 0,C 180,E1 -10063.404,E2 -10063.404} C_VEL
LIN {X 0,Y 418.342,Z 327.375,A -85,B 0,C 180,E1 -10066.999,E2 -10066.999} C_VEL
LIN {X 0,Y 418.337,Z 327.377,A -85,B 0,C 180,E1 -10070.328,E2 -10070.328} C_VEL
LIN {X 0,Y 418.509,Z 327.355,A -85,B 0,C 180,E1 -10072.279,E2 -10072.279} C_VEL
LIN {X 0,Y 418.51,Z 327.354,A -85,B 0,C 180,E1 -10074.217,E2 -10074.217} C_VEL
LIN {X 0,Y 418.537,Z 327.35,A -85,B 0,C 180,E1 -10078.075,E2 -10078.075} C_VEL
LIN {X 0,Y 418.656,Z 327.336,A -85,B 0,C 180,E1 -10080,E2 -10080} C_VEL
LIN {X 0,Y 418.496,Z 327.355,A -85,B 0,C 180,E1 -10082.888,E2 -10082.888} C_VEL
LIN {X 0,Y 418.489,Z 327.356,A -85,B 0,C 180,E1 -10086.751,E2 -10086.751} C_VEL
LIN {X 0,Y 418.337,Z 327.375,A -85,B 0,C 180,E1 -10089.671,E2 -10089.671} C_VEL
LIN {X 0,Y 418.342,Z 327.371,A -85,B 0,C 180,E1 -10093.001,E2 -10093.001} C_VEL
LIN {X 0,Y 418.309,Z 327.377,A -85,B 0,C 180,E1 -10096.735,E2 -10096.735} C_VEL
LIN {X 0,Y 418.267,Z 327.385,A -85,B 0,C 180,E1 -10099.79,E2 -10099.79} C_VEL
LIN {X 0,Y 418.234,Z 327.386,A -85,B 0,C 180,E1 -10102.736,E2 -10102.736} C_VEL
LIN {X 0,Y 418.231,Z 327.389,A -85,B 0,C 180,E1 -10105.907,E2 -10105.907} C_VEL
LIN {X 0,Y 418.255,Z 327.386,A -85,B 0,C 180,E1 -10109.163,E2 -10109.163} C_VEL
LIN {X 0,Y 418.255,Z 327.385,A -85,B 0,C 180,E1 -10112.844,E2 -10112.844} C_VEL
LIN {X 0,Y 418.246,Z 327.385,A -85,B 0,C 180,E1 -10116.239,E2 -10116.239} C_VEL
LIN {X 0,Y 418.199,Z 327.391,A -85,B 0,C 180,E1 -10119.688,E2 -10119.688} C_VEL
LIN {X 0,Y 418.205,Z 327.389,A -85,B 0,C 180,E1 -10122.318,E2 -10122.318} C_VEL
LIN {X 0,Y 418.234,Z 327.39,A -85,B 0,C 180,E1 -10125.109,E2 -10125.109} C_VEL
LIN {X 0,Y 418.255,Z 327.387,A -85,B 0,C 180,E1 -10128.897,E2 -10128.897} C_VEL
LIN {X 0,Y 418.477,Z 328.584,A -85,B 0,C 180,E1 -10129.744,E2 -10129.744} C_VEL
LIN {X 0,Y 419.371,Z 334.074,A -85,B 0,C 180,E1 -10132.893,E2 -10132.893} C_VEL
LIN {X 0,Y 419.524,Z 338.516,A -85,B 0,C 180,E1 -10135.279,E2 -10135.279} C_VEL
LIN {X 0,Y 419.065,Z 345.438,A -85,B 0,C 180,E1 -10138.794,E2 -10138.794} C_VEL
LIN {X 0,Y 418.741,Z 350.799,A -85,B 0,C 180,E1 -10141.424,E2 -10141.424} C_VEL
LIN {X 0,Y 418.363,Z 357.527,A -85,B 0,C 180,E1 -10144.636,E2 -10144.636} C_VEL
LIN {X 0,Y 418.042,Z 363.856,A -85,B 0,C 180,E1 -10147.615,E2 -10147.615} C_VEL
LIN {X 0,Y 417.764,Z 370.876,A -85,B 0,C 180,E1 -10150.872,E2 -10150.872} C_VEL
LIN {X 0,Y 417.616,Z 374.971,A -85,B 0,C 180,E1 -10152.729,E2 -10152.729} C_VEL
LIN {X 0,Y 420.074,Z 388.445,A -85,B 0,C 180,E1 -10153.237,E2 -10153.237} C_VEL
LIN {X 0,Y 421.873,Z 400.451,A -85,B 0,C 180,E1 -10153.859,E2 -10153.859} C_VEL
LIN {X 0,Y 421.16,Z 413.303,A -85,B 0,C 180,E1 -10154.638,E2 -10154.638} C_VEL
LIN {X 0,Y 420.528,Z 423.989,A -85,B 0,C 180,E1 -10155.482,E2 -10155.482} C_VEL
LIN {X 0,Y 419.766,Z 434.902,A -85,B 0,C 180,E1 -10156.567,E2 -10156.567} C_VEL
LIN {X 0,Y 419.159,Z 443.805,A -85,B 0,C 180,E1 -10157.656,E2 -10157.656} C_VEL
LIN {X 0,Y 418.42,Z 453.477,A -85,B 0,C 180,E1 -10159.108,E2 -10159.108} C_VEL
LIN {X 0,Y 417.904,Z 461.18,A -85,B 0,C 180,E1 -10160.562,E2 -10160.562} C_VEL
LIN {X 0,Y 417.413,Z 468.28,A -85,B 0,C 180,E1 -10162.259,E2 -10162.259} C_VEL
LIN {X 0,Y 417.226,Z 472.771,A -85,B 0,C 180,E1 -10163.634,E2 -10163.634} C_VEL
LIN {X 0,Y 417.151,Z 476.622,A -85,B 0,C 180,E1 -10165.167,E2 -10165.167} C_VEL
LIN {X 0,Y 417.023,Z 478.484,A -85,B 0,C 180,E1 -10166.134,E2 -10166.134} C_VEL
LIN {X 0,Y 417.024,Z 479.883,A -85,B 0,C 180,E1 -10167.102,E2 -10167.102} C_VEL
LIN {X 0,Y 417.053,Z 480.882,A -85,B 0,C 180,E1 -10168.068,E2 -10168.068} C_VEL
LIN {X 0,Y 416.992,Z 481.489,A -85,B 0,C 180,E1 -10169.034,E2 -10169.034} C_VEL
LIN {X 0,Y 416.963,Z 481.705,A -85,B 0,C 180,E1 -10170,E2 -10170} C_VEL
LIN {X 0,Y 417.052,Z 480.884,A -85,B 0,C 180,E1 -10171.931,E2 -10171.931} C_VEL
LIN {X 0,Y 417.023,Z 479.887,A -85,B 0,C 180,E1 -10172.898,E2 -10172.898} C_VEL
LIN {X 0,Y 417.023,Z 478.489,A -85,B 0,C 180,E1 -10173.865,E2 -10173.865} C_VEL
LIN {X 0,Y 417.164,Z 475.553,A -85,B 0,C 180,E1 -10175.316,E2 -10175.316} C_VEL
LIN {X 0,Y 417.275,Z 471.575,A -85,B 0,C 180,E1 -10176.77,E2 -10176.77} C_VEL
LIN {X 0,Y 417.628,Z 465.464,A -85,B 0,C 180,E1 -10178.467,E2 -10178.467} C_VEL
LIN {X 0,Y 418.043,Z 458.784,A -85,B 0,C 180,E1 -10179.922,E2 -10179.922} C_VEL
LIN {X 0,Y 418.615,Z 450.499,A -85,B 0,C 180,E1 -10181.377,E2 -10181.377} C_VEL
LIN {X 0,Y 419.339,Z 442.013,A -85,B 0,C 180,E1 -10182.584,E2 -10182.584} C_VEL
LIN {X 0,Y 420.065,Z 431.583,A -85,B 0,C 180,E1 -10183.786,E2 -10183.786} C_VEL
LIN {X 0,Y 420.665,Z 421.147,A -85,B 0,C 180,E1 -10184.76,E2 -10184.76} C_VEL
LIN {X 0,Y 421.419,Z 409.776,A -85,B 0,C 180,E1 -10185.599,E2 -10185.599} C_VEL
LIN {X 0,Y 421.81,Z 400.454,A -85,B 0,C 180,E1 -10186.142,E2 -10186.142} C_VEL
LIN {X 0,Y 419.87,Z 387.223,A -85,B 0,C 180,E1 -10186.817,E2 -10186.817} C_VEL
LIN {X 0,Y 417.607,Z 374.844,A -85,B 0,C 180,E1 -10187.291,E2 -10187.291} C_VEL
LIN {X 0,Y 417.897,Z 367.528,A -85,B 0,C 180,E1 -10190.68,E2 -10190.68} C_VEL
LIN {X 0,Y 418.249,Z 359.761,A -85,B 0,C 180,E1 -10194.31,E2 -10194.31} C_VEL
LIN {X 0,Y 418.565,Z 353.773,A -85,B 0,C 180,E1 -10197.138,E2 -10197.138} C_VEL
LIN {X 0,Y 418.953,Z 347.42,A -85,B 0,C 180,E1 -10200.214,E2 -10200.214} C_VEL
LIN {X 0,Y 419.341,Z 340.724,A -85,B 0,C 180,E1 -10203.576,E2 -10203.576} C_VEL
LIN {X 0,Y 419.512,Z 336.286,A -85,B 0,C 180,E1 -10205.897,E2 -10205.897} C_VEL
LIN {X 0,Y 419.051,Z 331.839,A -85,B 0,C 180,E1 -10208.354,E2 -10208.354} C_VEL
LIN {X 0,Y 418.298,Z 327.385,A -85,B 0,C 180,E1 -10211.017,E2 -10211.017} C_VEL
LIN {X 0,Y 418.279,Z 327.389,A -85,B 0,C 180,E1 -10213.739,E2 -10213.739} C_VEL
LIN {X 0,Y 418.196,Z 327.393,A -85,B 0,C 180,E1 -10216.447,E2 -10216.447} C_VEL
LIN {X 0,Y 418.204,Z 327.391,A -85,B 0,C 180,E1 -10219.131,E2 -10219.131} C_VEL
LIN {X 0,Y 418.221,Z 327.389,A -85,B 0,C 180,E1 -10222.166,E2 -10222.166} C_VEL
LIN {X 0,Y 418.259,Z 327.383,A -85,B 0,C 180,E1 -10225.419,E2 -10225.419} C_VEL
LIN {X 0,Y 418.203,Z 327.394,A -85,B 0,C 180,E1 -10228.603,E2 -10228.603} C_VEL
LIN {X 0,Y 418.211,Z 327.39,A -85,B 0,C 180,E1 -10231.931,E2 -10231.931} C_VEL
LIN {X 0,Y 418.263,Z 327.382,A -85,B 0,C 180,E1 -10235.161,E2 -10235.161} C_VEL
LIN {X 0,Y 418.225,Z 327.391,A -85,B 0,C 180,E1 -10238.303,E2 -10238.303} C_VEL
LIN {X 0,Y 418.274,Z 327.382,A -85,B 0,C 180,E1 -10241.383,E2 -10241.383} C_VEL
LIN {X 0,Y 418.29,Z 327.382,A -85,B 0,C 180,E1 -10244.405,E2 -10244.405} C_VEL
LIN {X 0,Y 418.345,Z 327.372,A -85,B 0,C 180,E1 -10247.385,E2 -10247.385} C_VEL
LIN {X 0,Y 418.331,Z 327.376,A -85,B 0,C 180,E1 -10250.328,E2 -10250.328} C_VEL
LIN {X 0,Y 418.487,Z 327.356,A -85,B 0,C 180,E1 -10253.249,E2 -10253.249} C_VEL
LIN {X 0,Y 418.337,Z 327.374,A -85,B 0,C 180,E1 -10255.182,E2 -10255.182} C_VEL
LIN {X 0,Y 418.533,Z 327.352,A -85,B 0,C 180,E1 -10258.075,E2 -10258.075} C_VEL
LIN {X 0,Y 418.652,Z 327.337,A -85,B 0,C 180,E1 -10260,E2 -10260} C_VEL
LIN {X 0,Y 418.492,Z 327.353,A -85,B 0,C 180,E1 -10262.888,E2 -10262.888} C_VEL
LIN {X 0,Y 418.485,Z 327.355,A -85,B 0,C 180,E1 -10266.751,E2 -10266.751} C_VEL
LIN {X 0,Y 418.331,Z 327.378,A -85,B 0,C 180,E1 -10269.672,E2 -10269.672} C_VEL
LIN {X 0,Y 418.336,Z 327.376,A -85,B 0,C 180,E1 -10273.001,E2 -10273.001} C_VEL
LIN {X 0,Y 418.303,Z 327.378,A -85,B 0,C 180,E1 -10276.736,E2 -10276.736} C_VEL
LIN {X 0,Y 418.262,Z 327.384,A -85,B 0,C 180,E1 -10279.791,E2 -10279.791} C_VEL
LIN {X 0,Y 418.229,Z 327.39,A -85,B 0,C 180,E1 -10282.737,E2 -10282.737} C_VEL
LIN {X 0,Y 418.226,Z 327.387,A -85,B 0,C 180,E1 -10285.907,E2 -10285.907} C_VEL
LIN {X 0,Y 418.25,Z 327.387,A -85,B 0,C 180,E1 -10289.163,E2 -10289.163} C_VEL
LIN {X 0,Y 418.25,Z 327.388,A -85,B 0,C 180,E1 -10292.845,E2 -10292.845} C_VEL
LIN {X 0,Y 418.239,Z 327.387,A -85,B 0,C 180,E1 -10296.239,E2 -10296.239} C_VEL
LIN {X 0,Y 418.194,Z 327.391,A -85,B 0,C 180,E1 -10299.689,E2 -10299.689} C_VEL
LIN {X 0,Y 418.205,Z 327.392,A -85,B 0,C 180,E1 -10302.319,E2 -10302.319} C_VEL
LIN {X 0,Y 418.23,Z 327.386,A -85,B 0,C 180,E1 -10305.11,E2 -10305.11} C_VEL
LIN {X 0,Y 418.252,Z 327.384,A -85,B 0,C 180,E1 -10307.77,E2 -10307.77} C_VEL
LIN {X 0,Y 418.262,Z 327.386,A -85,B 0,C 180,E1 -10310.618,E2 -10310.618} C_VEL
LIN {X 0,Y 418.148,Z 327.401,A -85,B 0,C 180,E1 -10313.968,E2 -10313.968} C_VEL
LIN {X 0,Y 418.154,Z 329.968,A -85,B 0,C 180,E1 -10316.315,E2 -10316.315} C_VEL
LIN {X 0,Y 417.93,Z 334.253,A -85,B 0,C 180,E1 -10319.704,E2 -10319.704} C_VEL
LIN {X 0,Y 417.758,Z 338.628,A -85,B 0,C 180,E1 -10323.079,E2 -10323.079} C_VEL
LIN {X 0,Y 417.595,Z 342.755,A -85,B 0,C 180,E1 -10326.178,E2 -10326.178} C_VEL
LIN {X 0,Y 417.442,Z 347.07,A -85,B 0,C 180,E1 -10329.296,E2 -10329.296} C_VEL
LIN {X 0,Y 417.351,Z 351.471,A -85,B 0,C 180,E1 -10332.356,E2 -10332.356} C_VEL
LIN {X 0,Y 417.374,Z 352.265,A -85,B 0,C 180,E1 -10332.799,E2 -10332.799} C_VEL
LIN {X 0,Y 420.545,Z 365.651,A -85,B 0,C 180,E1 -10333.371,E2 -10333.371} C_VEL
LIN {X 0,Y 422.217,Z 374.753,A -85,B 0,C 180,E1 -10333.861,E2 -10333.861} C_VEL
LIN {X 0,Y 421.667,Z 386.217,A -85,B 0,C 180,E1 -10334.534,E2 -10334.534} C_VEL
LIN {X 0,Y 421.005,Z 397.319,A -85,B 0,C 180,E1 -10335.376,E2 -10335.376} C_VEL
LIN {X 0,Y 420.347,Z 408.628,A -85,B 0,C 180,E1 -10336.464,E2 -10336.464} C_VEL
LIN {X 0,Y 419.534,Z 418.606,A -85,B 0,C 180,E1 -10337.668,E2 -10337.668} C_VEL
LIN {X 0,Y 418.822,Z 428.247,A -85,B 0,C 180,E1 -10339.119,E2 -10339.119} C_VEL
LIN {X 0,Y 418.23,Z 435.939,A -85,B 0,C 180,E1 -10340.571,E2 -10340.571} C_VEL
LIN {X 0,Y 417.693,Z 442.996,A -85,B 0,C 180,E1 -10342.265,E2 -10342.265} C_VEL
LIN {X 0,Y 417.491,Z 447.366,A -85,B 0,C 180,E1 -10343.606,E2 -10343.606} C_VEL
LIN {X 0,Y 417.23,Z 451.292,A -85,B 0,C 180,E1 -10345.169,E2 -10345.169} C_VEL
LIN {X 0,Y 417.152,Z 453.151,A -85,B 0,C 180,E1 -10346.136,E2 -10346.136} C_VEL
LIN {X 0,Y 417.158,Z 454.549,A -85,B 0,C 180,E1 -10347.103,E2 -10347.103} C_VEL
LIN {X 0,Y 417.014,Z 456.16,A -85,B 0,C 180,E1 -10349.035,E2 -10349.035} C_VEL
LIN {X 0,Y 417.004,Z 456.394,A -85,B 0,C 180,E1 -10350,E2 -10350} C_VEL
LIN {X 0,Y 417.014,Z 456.202,A -85,B 0,C 180,E1 -10350.972,E2 -10350.972} C_VEL
LIN {X 0,Y 417.158,Z 454.654,A -85,B 0,C 180,E1 -10352.897,E2 -10352.897} C_VEL
LIN {X 0,Y 417.148,Z 453.301,A -85,B 0,C 180,E1 -10353.864,E2 -10353.864} C_VEL
LIN {X 0,Y 417.28,Z 450.898,A -85,B 0,C 180,E1 -10355.104,E2 -10355.104} C_VEL
LIN {X 0,Y 416.762,Z 449.117,A -85,B 0,C 180,E1 -10355.873,E2 -10355.873} C_VEL
LIN {X 0,Y 414.094,Z 445.781,A -85,B 0,C 180,E1 -10357.106,E2 -10357.106} C_VEL
LIN {X 0,Y 411.455,Z 441.846,A -85,B 0,C 180,E1 -10358.318,E2 -10358.318} C_VEL
LIN {X 0,Y 410.999,Z 439.011,A -85,B 0,C 180,E1 -10359.045,E2 -10359.045} C_VEL
LIN {X 0,Y 411.559,Z 431.715,A -85,B 0,C 180,E1 -10360.578,E2 -10360.578} C_VEL
LIN {X 0,Y 412.289,Z 422.905,A -85,B 0,C 180,E1 -10362.053,E2 -10362.053} C_VEL
LIN {X 0,Y 413.061,Z 413.862,A -85,B 0,C 180,E1 -10363.279,E2 -10363.279} C_VEL
LIN {X 0,Y 413.725,Z 404.086,A -85,B 0,C 180,E1 -10364.362,E2 -10364.362} C_VEL
LIN {X 0,Y 414.432,Z 392.716,A -85,B 0,C 180,E1 -10365.365,E2 -10365.365} C_VEL
LIN {X 0,Y 415.157,Z 380.757,A -85,B 0,C 180,E1 -10366.185,E2 -10366.185} C_VEL
LIN {X 0,Y 415.208,Z 374.622,A -85,B 0,C 180,E1 -10366.536,E2 -10366.536} C_VEL
LIN {X 0,Y 412.757,Z 362.588,A -85,B 0,C 180,E1 -10367.181,E2 -10367.181} C_VEL
LIN {X 0,Y 410.257,Z 352.298,A -85,B 0,C 180,E1 -10367.625,E2 -10367.625} C_VEL
LIN {X 0,Y 410.368,Z 348.852,A -85,B 0,C 180,E1 -10370.031,E2 -10370.031} C_VEL
LIN {X 0,Y 410.49,Z 344.528,A -85,B 0,C 180,E1 -10373.19,E2 -10373.19} C_VEL
LIN {X 0,Y 410.606,Z 341.633,A -85,B 0,C 180,E1 -10375.335,E2 -10375.335} C_VEL
LIN {X 0,Y 410.776,Z 337.387,A -85,B 0,C 180,E1 -10378.624,E2 -10378.624} C_VEL
LIN {X 0,Y 411.012,Z 333.121,A -85,B 0,C 180,E1 -10382.01,E2 -10382.01} C_VEL
LIN {X 0,Y 411.128,Z 329.606,A -85,B 0,C 180,E1 -10384.861,E2 -10384.861} C_VEL
LIN {X 0,Y 411.099,Z 328.791,A -85,B 0,C 180,E1 -10385.538,E2 -10385.538} C_VEL
LIN {X 0,Y 411.163,Z 328.274,A -85,B 0,C 180,E1 -10386.745,E2 -10386.745} C_VEL
LIN {X 0,Y 411.208,Z 328.265,A -85,B 0,C 180,E1 -10389.727,E2 -10389.727} C_VEL
LIN {X 0,Y 411.173,Z 328.267,A -85,B 0,C 180,E1 -10393.133,E2 -10393.133} C_VEL
LIN {X 0,Y 411.162,Z 328.269,A -85,B 0,C 180,E1 -10395.881,E2 -10395.881} C_VEL
LIN {X 0,Y 411.156,Z 328.272,A -85,B 0,C 180,E1 -10399.493,E2 -10399.493} C_VEL
LIN {X 0,Y 411.185,Z 328.265,A -85,B 0,C 180,E1 -10402.025,E2 -10402.025} C_VEL
LIN {X 0,Y 411.204,Z 328.264,A -85,B 0,C 180,E1 -10405.666,E2 -10405.666} C_VEL
LIN {X 0,Y 411.186,Z 328.269,A -85,B 0,C 180,E1 -10409.152,E2 -10409.152} C_VEL
LIN {X 0,Y 411.175,Z 328.268,A -85,B 0,C 180,E1 -10411.407,E2 -10411.407} C_VEL
LIN {X 0,Y 411.213,Z 328.265,A -85,B 0,C 180,E1 -10414.932,E2 -10414.932} C_VEL
LIN {X 0,Y 411.202,Z 328.262,A -85,B 0,C 180,E1 -10417.913,E2 -10417.913} C_VEL
LIN {X 0,Y 411.221,Z 328.264,A -85,B 0,C 180,E1 -10421.051,E2 -10421.051} C_VEL
LIN {X 0,Y 411.249,Z 328.255,A -85,B 0,C 180,E1 -10424.131,E2 -10424.131} C_VEL
LIN {X 0,Y 411.299,Z 328.252,A -85,B 0,C 180,E1 -10427.165,E2 -10427.165} C_VEL
LIN {X 0,Y 411.289,Z 328.253,A -85,B 0,C 180,E1 -10430.161,E2 -10430.161} C_VEL
LIN {X 0,Y 411.478,Z 328.23,A -85,B 0,C 180,E1 -10432.147,E2 -10432.147} C_VEL
LIN {X 0,Y 411.472,Z 328.231,A -85,B 0,C 180,E1 -10434.118,E2 -10434.118} C_VEL
LIN {X 0,Y 411.506,Z 328.226,A -85,B 0,C 180,E1 -10438.042,E2 -10438.042} C_VEL
LIN {X 0,Y 411.626,Z 328.211,A -85,B 0,C 180,E1 -10440,E2 -10440} C_VEL
LIN {X 0,Y 411.453,Z 328.231,A -85,B 0,C 180,E1 -10442.937,E2 -10442.937} C_VEL
LIN {X 0,Y 411.471,Z 328.232,A -85,B 0,C 180,E1 -10445.882,E2 -10445.882} C_VEL
LIN {X 0,Y 411.35,Z 328.243,A -85,B 0,C 180,E1 -10448.845,E2 -10448.845} C_VEL
LIN {X 0,Y 411.279,Z 328.255,A -85,B 0,C 180,E1 -10451.833,E2 -10451.833} C_VEL
LIN {X 0,Y 411.252,Z 328.255,A -85,B 0,C 180,E1 -10454.853,E2 -10454.853} C_VEL
LIN {X 0,Y 411.248,Z 328.26,A -85,B 0,C 180,E1 -10457.915,E2 -10457.915} C_VEL
LIN {X 0,Y 411.193,Z 328.264,A -85,B 0,C 180,E1 -10461.034,E2 -10461.034} C_VEL
LIN {X 0,Y 411.214,Z 328.261,A -85,B 0,C 180,E1 -10464.216,E2 -10464.216} C_VEL
LIN {X 0,Y 411.175,Z 328.27,A -85,B 0,C 180,E1 -10467.484,E2 -10467.484} C_VEL
LIN {X 0,Y 411.194,Z 328.266,A -85,B 0,C 180,E1 -10469.713,E2 -10469.713} C_VEL
LIN {X 0,Y 411.204,Z 328.266,A -85,B 0,C 180,E1 -10473.156,E2 -10473.156} C_VEL
LIN {X 0,Y 411.193,Z 328.263,A -85,B 0,C 180,E1 -10476.553,E2 -10476.553} C_VEL
